                MoveJ Offs(ptPolish,0,0,500),v500,z5,tPolish;
            ENDIF

        DEFAULT:
            !Unknown
            RAISE ERR_TC_SELECTION;

        ENDTEST
        IF dropoffTool THEN
        MoveJ pHome,vMax,fine,tTCMaster;
        ENDIF

    ERROR
        RAISE ;

    ENDPROC

    FUNC num PointToPointDist(num px,num py,num x1,num y1)
        !Used to check if point is within helicopter blades

        VAR num Dist;

        Dist:=Sqrt((x1-px)*(x1-px)+(y1-py)*(y1-py));
        RETURN Dist;
    ENDFUNC

    FUNC num HighestArray(num count)
        !Used to determine highest height offset
        VAR num j;
        VAR num HighestValue;
        HighestValue:=HeliZArray{1};
        FOR j FROM 1 TO count DO
            IF HeliZArray{j}>HighestValue THEN
                HighestValue:=HeliZArray{j};
            ENDIF
        ENDFOR
        IF PreviousHighest>HighestValue THEN
            PreviousHighest:=HighestValue;
            RETURN PreviousHighest;
        ELSEIF HighestValue<=-30 THEN
            PreviousHighest:=HighestValue;
            RETURN 0;
        ELSE
            PreviousHighest:=HighestValue;
            RETURN HighestValue;
        ENDIF

    ENDFUNC

    PROC HeliZ(num x1,num y1,bool ResetZArray)
        !Determines height offsets for helicopter movements
        VAR num CloseYPos;
        x1:=Abs(x1);
        IF ResetZArray=TRUE THEN
            HeliZArrayCounter:=1;
            FOR i FROM 1 TO DIM(HeliZArray,1) DO
                HeliZArray{i}:=-50;
            ENDFOR
        ENDIF

        FOR i FROM 1 TO 17 DO
            FOR j FROM 1 TO 4 DO
                IF PointToPointDist(x1,y1,BedZpos{j,i,1},BedZpos{j,i,2})<=HeliBladeWidth/2 THEN
                    HeliZArray{HeliZArrayCounter}:=BedZreads{j,i};
                    Incr HeliZArrayCounter;
                ENDIF
            ENDFOR
        ENDFOR

    ENDPROC

    PROC PlotBedGrid(num Xcord1,num Ycord1,num ZOffset)
        !Used by BedGridPlotter for Z datum
        Plotterp1.trans:=[Xcord1,Ycord1,200+ZOffset];
        !+46

        IF Plotterp1.trans.y>0 THEN
            IF Plotterp1.trans.y<(abs(tPlotter.tframe.trans.x)-10) THEN
                PlotterZOri:=ACos(Plotterp1.trans.y/abs(tPlotter.tframe.trans.x));
                IF PlotterZOri>PlotA6Max THEN
                    PlotterZOri:=90;
                ENDIF
                Plotterp1.rot:=OrientZYX(-90+PlotterZOri,0,180);
            ELSE
                PlotterZOri:=0;
                Plotterp1.rot:=OrientZYX(-90,0,180);
            ENDIF
        ELSE
            RAISE ERR_PLOT_POS;
        ENDIF

        IF PlotterP1.trans.y>(abs(tPlotter.tframe.trans.x)+250) THEN
            Plotterp1.extax:=[(Plotterp1.trans.x+Bed1.uframe.trans.x),9E+09,9E+09,9E+09,9E+09,9E+09];
        ELSE
            Plotterp1.extax:=[(Plotterp1.trans.x+Bed1.uframe.trans.x+1000+Abs(tPlotter.tframe.trans.x*Sin(PlotterZOri))),9E+09,9E+09,9E+09,9E+09,9E+09];
        ENDIF

        IF Plotterp1.extax.eax_a>10150 THEN
            Plotterp1.extax.eax_a:=10100;
        ENDIF

        IF Plotterp1.extax.eax_a<0 THEN
            Plotterp1.extax.eax_a:=0;
        ENDIF

        vPlotter:=[100,15,2000,15];

        MoveL Plotterp1,v300,zPlotter,tTCMaster\WObj:=Bed1Wyong;

    ENDPROC

    PROC BedGridPlotter()
        !Get Z datum offset
        FOR k FROM 7 TO 19 DO
            !Move x
            FOR j FROM 4 TO 9 DO
                !Move y

                PlotBedGrid(k*XGridSpacing+100),(j*YGridSpacing+100),Bed1Zread{10-j,(k+1)};
                WaitTime\inpos,0.1;

            ENDFOR

        ENDFOR

    ENDPROC

    PROC MoveGridDatum()
        !Sweep across bed maintaining Z height through offsets
        FOR j FROM 9 TO 4 DO
            FOR k FROM 11 TO 1 DO
                !Move x
                PlotBedGrid(k*XGridSpacing+100),(j*YGridSpacing+100),Bed1Zread{10-j,(k+1)};
            ENDFOR
        ENDFOR
    ENDPROC


    PROC VacuumBed()

        VAR num VacOverlap:=-400;
        UpdateToolNum;
        IF ToolNum<>5 THEN
            Home TRUE;
            Vac_Pickup;
        ELSE
            CurrentJoints:=CJointT();
            CurrentPos:=CalcRobT(CurrentJoints,tVac\WObj:=Bed1Wyong);
            IF CurrentPos.trans.x<0 AND (CurrentPos.trans.z<150) THEN
                MoveL Offs(CurrentPos,0,0,(150-CurrentPos.trans.z)),v500,z5,tVac\WObj:=Bed1Wyong;
            ELSEIF (CurrentPos.trans.z<700) THEN
                MoveL Offs(CurrentPos,0,0,(700-CurrentPos.trans.z)),v500,z5,tVac\WObj:=Bed1Wyong;
            ENDIF
        ENDIF

        pTemp:=pVacStart;
        pTemp2:=pVacStart;
        pTemp2.trans.x:=pVacStart2.trans.x;
        pTemp2.extax.eax_a:=pVacStart2.extax.eax_a;

        Vac_on;
        FOR i FROM 0 TO (Round((pVacStart.trans.y-pVacStart2.trans.y)/(-1*VacOverlap))) DO
            IF pTemp.trans.y+i*VacOverlap>pVacStart2.trans.y THEN
                MoveJ Offs(pTemp,0,i*VacOverlap,150),v500,z5,tVac\WObj:=Bed1Wyong;
                MoveL Offs(pTemp,0,i*VacOverlap,0),v50,z5,tVac\WObj:=Bed1Wyong;
                MoveL Offs(pTemp2,0,i*VacOverlap,0),v100,z5,tVac\WObj:=Bed1Wyong;
                MoveL Offs(pTemp2,0,i*VacOverlap,150),v50,fine,tVac\WObj:=Bed1Wyong;
            ENDIF
        ENDFOR

        Vac_off;

        CurrentJoints:=CJointT();
        CurrentPos:=CalcRobT(CurrentJoints,tVac\WObj:=wobj0);
        MoveL Offs(CurrentPos,0,0,800-CurrentPos.trans.z),v100,z5,tVac\WObj:=wobj0;

    ENDPROC

    PROC JointPositions()

        VAR num PolishOverlap:=450;
        pPolTemp:=pPolStart1;
        pPolTemp2:=pPolStart1;
        pPolTemp2.extax.eax_a:=pPolStart1.extax.eax_a-7500;
        pPolTemp2.trans.x:=-7500;

        pPolTemp.rot:=pPolStart1.rot;
        pPolTemp2.rot:=pPolStart1.rot;

        pPolTemp2.rot:=pPolStart2.rot;
        pPolTemp2.extax.eax_a:=pPolStart1.extax.eax_a-8500;
        CurrentJoints5:=CJointT();
        CurrentJoints6:=CalcJointT(Offs(pPolTemp2,50,(1+1)*PolishOverlap,40),tPolish\WObj:=Bed1Wyong);

    ENDPROC


    PROC RobbiePlot()

        ! !Write R
        !PlotLine 6900,1000, 6900,2000;
        !PlotArc 6900,2000,6650,1750,6900,1500;
        !PlotLine 6900,1500,6650,1000;

        !!Write O
        !PlotArc 6300,2000, 6050,1500,6300,1000;
        !PlotArc 6300,1000, 6550,1500,6300,2000;

        !!Write B
        !PlotLine 5700,1000, 5700,2000;
        !PlotArc 5700,2000,5450,1750,5700,1500;
        !PlotArc 5700,1500,5450,1250,5700,1000;

        !!Write B
        !PlotLine 5100,1000, 5100,2000;
        !PlotArc 5100,2000,4850,1750,5100,1500;
        !PlotArc 5100,1500,4850,1250,5100,1000;

        !!Write I
        !PlotLine 4500,1000, 4500,2000;

        !!Write E
        !PlotLine 3900,1000, 3900,2000;
        !PlotLine 3900,2000, 3400,2000;
        !PlotLine 3900,1500, 3400,1500;
        !PlotLine 3900,1000, 3400,1000;

        !formbox
        PlotRect 2000,500,2000,3500,6000,3500,6000,500;
        !Ferrule
        WaitTime\inpos,0.1;
        PlotCirc 2250,750,(PlotCircleD/2);
        PlotLine(2250-PlotCircleD/2-CrossHairExt),750,(2250+PlotCircleD/2+CrossHairExt),750;
        PlotLine 2250,(750-PlotCircleD/2-CrossHairExt),2250,(750+PlotCircleD/2+CrossHairExt);
        !Ferrule
        WaitTime\inpos,0.1;
        PlotCirc 2250,3250,(PlotCircleD/2);
        PlotLine(2250-PlotCircleD/2-CrossHairExt),3250,(2250+PlotCircleD/2+CrossHairExt),3250;
        PlotLine 2250,(3250-PlotCircleD/2-CrossHairExt),2250,(3250+PlotCircleD/2+CrossHairExt);
        !Grout tube Casee 4
        WaitTime\inpos,0.1;
        iCoord1x:=6000;
        iCoord1y:=2000;
        iAngle:=0;
        PlotRect iCoord1x-GroutWidth/2*Sin(iAngle)-GroutHeight*Cos(iAngle),iCoord1y+GroutHeight*Sin(iAngle)-GroutWidth/2*Cos(iAngle),iCoord1x+GroutWidth/2*Sin(iAngle)-GroutHeight*Cos(iAngle),iCoord1y+GroutHeight*Sin(iAngle)+GroutWidth/2*Cos(iAngle),iCoord1x+GroutWidth/2*Sin(iAngle),iCoord1y+GroutWidth/2*Cos(iAngle),iCoord1x-GroutWidth/2*Sin(iAngle),iCoord1y-GroutWidth/2*Cos(iAngle);

        !Lifting points 180 angle
        WaitTime\inpos,0.1;
        TriangleAngle:=180;
        iCoord1x:=5000;
        iCoord1y:=3500;
        PlotLine iCoord1x-TriangleHeight*Sin(TriangleAngle),iCoord1y-TriangleHeight*Cos(TriangleAngle),iCoord1x-TriangleBase/2*Cos(TriangleAngle),iCoord1y+TriangleBase/2*Sin(TriangleAngle);
        PlotLine iCoord1x-TriangleBase/2*Cos(TriangleAngle),iCoord1y+TriangleBase/2*Sin(TriangleAngle),iCoord1x+TriangleBase/2*Cos(TriangleAngle),iCoord1y-TriangleBase/2*Sin(TriangleAngle);
        PlotLine iCoord1x+TriangleBase/2*Cos(TriangleAngle),iCoord1y-TriangleBase/2*Sin(TriangleAngle),iCoord1x-TriangleHeight*Sin(TriangleAngle),iCoord1y-TriangleHeight*Cos(TriangleAngle);
        !Lifting points 180 angle
        WaitTime\inpos,0.1;
        TriangleAngle:=180;
        iCoord1x:=3000;
        iCoord1y:=3500;
        PlotLine iCoord1x-TriangleHeight*Sin(TriangleAngle),iCoord1y-TriangleHeight*Cos(TriangleAngle),iCoord1x-TriangleBase/2*Cos(TriangleAngle),iCoord1y+TriangleBase/2*Sin(TriangleAngle);
        PlotLine iCoord1x-TriangleBase/2*Cos(TriangleAngle),iCoord1y+TriangleBase/2*Sin(TriangleAngle),iCoord1x+TriangleBase/2*Cos(TriangleAngle),iCoord1y-TriangleBase/2*Sin(TriangleAngle);
        PlotLine iCoord1x+TriangleBase/2*Cos(TriangleAngle),iCoord1y-TriangleBase/2*Sin(TriangleAngle),iCoord1x-TriangleHeight*Sin(TriangleAngle),iCoord1y-TriangleHeight*Cos(TriangleAngle);

        Plotter_Dropoff;

    ENDPROC

    PROC PolishDemo()
        UpdateToolNum;
        IF ToolNum<>6 THEN
            Home TRUE;
            Polish_Pickup;
        ELSE
            CurrentJoints:=CJointT();
            CurrentPos:=CalcRobT(CurrentJoints,tPolish\WObj:=wobj0);
            IF CurrentPos.trans.z<600 THEN
                MoveL Offs(CurrentPos,0,0,(600-CurrentPos.trans.z)),v500,z5,tPolish;
            ENDIF
        ENDIF
        MoveJ pPolHome,v500,z5,tPolish;
        pPolTemp:=pPolStart1;
        pPolTemp2:=pPolStart1;
        pPolTemp2.extax.eax_a:=pPolStart1.extax.eax_a-7500;
        pPolTemp2.trans.x:=-7500;
        pPolTemp.rot:=pPolStart1.rot;
        pPolTemp2.rot:=pPolStart1.rot;
        FCCalib PolishLoad;
        pPolTemp.extax.eax_a:=pPolStart1.extax.eax_a;
        MoveJ Offs(pPolTemp,0,0,100),v500,z5,tPolish\WObj:=Bed1Wyong;
        Pol_on;
        MoveL Offs(pPolTemp,0,0,50),v100,fine,tPolish\WObj:=Bed1Wyong;
        myForceVector:=FCGetForce(\Tool:=tPolish);
        FCPress1LStart Offs(pPolTemp,-25,0,55),v10,\Fz:=120,15,\ForceChange:=50\PosSupvDist:=125,z5,tPolish\WObj:=Bed1Wyong;
        pPolTemp2.extax.eax_a:=pPolStart2.extax.eax_a-300;
        FCPressL Offs(pPolTemp2,-300,0,-15),v100,130,fine,tPolish\WObj:=Bed1Wyong;
        FCPressEnd Offs(pPolTemp2,-300,0,75),v50,\DeactOnly,tPolish\WObj:=Bed1Wyong;
        CurrentJoints:=CJointT();
        CurrentPos:=CalcRobT(CurrentJoints,tPolish\WObj:=Bed1Wyong);
        MoveJ Offs(Reltool(CurrentPos,0,0,-100),0,450,0),v100,fine,tPolish\WObj:=Bed1Wyong;
        Pol_off;
        Polish_Dropoff;
    ENDPROC



    PROC BedGrid()

        !        MoveJ Offs(p10Maps,500*(1-1)+2000*(1-1),650*(1-1),50),v500,z5,tTCMaster\WObj:=Bed1Wyong;
        !        MoveL Offs(p10Maps,500*(1-1)+2000*(1-1),650*(1-1),0),v500,fine,tTCMaster\WObj:=Bed1Wyong;
        !        Stop;
        !        MoveL Offs(p10Maps,500*(1-1)+2000*(1-1),650*(1-1),50),v500,z5,tTCMaster\WObj:=Bed1Wyong;
        !        Stop;

        FOR i FROM 1 TO 5 DO
            !Move EAX
            FOR k FROM 1 TO 4 DO
                !Move x
                FOR j FROM 1 TO 4 DO
                    !Move y
                    IF 500*(k-1)+2000*(i-1)<8001 THEN
                        p10maps.extax.eax_a:=Bed1Wyong.uframe.trans.x+p10Maps.trans.x-500*(k-1)-2000*(i-1);
                        IF p10maps.extax.eax_a>10150 THEN
                            p10maps.extax.eax_a:=10100;
                        ENDIF
                        IF p10maps.extax.eax_a<1000 THEN
                            p10maps.extax.eax_a:=1000;
                        ENDIF

                        !MoveJ Offs(p10Maps,-500*(k-1)-2000*(i-1),650*(j-1),50),v500,z5,tTCMaster\WObj:=Bed1Wyong;
                        !MoveL Offs(p10Maps,-500*(k-1)-2000*(i-1),650*(j-1),0),v500,fine,tTCMaster\WObj:=Bed1Wyong;
                        !TPReadNum BedZread,"Enter Z reading";
                        !BedZreads{5-j,((i-1)*4+k)}:=BedZread;
                        BedZpos{5-j,((i-1)*4+k),1}:=p10Maps.trans.x-500*(k-1)-2000*(i-1);
                        BedZpos{5-j,((i-1)*4+k),2}:=p10maps.trans.y+650*(j-1);
                        !MoveL Offs(p10Maps,-500*(k-1)-2000*(i-1),650*(j-1),50),v500,z5,tTCMaster\WObj:=Bed1Wyong;
                    ENDIF

                ENDFOR
            ENDFOR
        ENDFOR
        Stop;

    ENDPROC


    PROC ClearBedZ()

        FOR i FROM 1 TO 4 DO
            !Move EAX
            FOR k FROM 1 TO 24 DO
                !Move x
                BedZreads{i,k}:=0;
                BedZpos{i,k,1}:=0;
                BedZpos{i,k,2}:=0;
            ENDFOR
        ENDFOR

    ENDPROC




    PROC BHTestTask()
        TPErase;
        TPWrite "BH Test Task";
        TPWrite "Press Play to confirm and start task";
        Stop;

        TPErase;
        TPWrite "Starting BH Test Task...";

        Heli_Pickup;
        MoveJ Offs(ptHeli,0,0,1000),v500,fine,tHeli;
        TPWrite "Helicopter tool at 1000mm above pickup";
        WaitTime 2;

        Heli_Dropoff;
        TPWrite "Helicopter tool dropped off";

        Polish_Pickup;
        MoveJ Offs(ptPolish,0,0,1000),v500,fine,tPolish;
        TPWrite "Polisher tool at 1000mm above pickup";
        WaitTime 2;

        Polish_Dropoff;
        TPWrite "Polisher tool dropped off";

        Home TRUE;
        TPWrite "BH Test Task Complete";

    ERROR
        RAISE ;
    ENDPROC



    PROC Datum()
        ! Datum - draws small circle at Bed1Wyong origin (0,0)
        ! Generated by Onyx Toolpath Generator
        VAR robtarget pDatumCenter;
        VAR robtarget pDatumCircle;
        VAR num DatumZ:=300;
        VAR num DatumRadius:=100;
        VAR num SafeZ:=500;
        VAR num i;

        UpdateToolNum;
        TPWrite "Datum: ToolNum=" \Num:=ToolNum;
        IF ToolNum<>4 THEN
            TPWrite "No plotter! Will pickup plotter.";
            Stop;
            Home TRUE;
            Plotter_Pickup;
        ELSE
            CurrentJoints:=CJointT();
            CurrentPos:=CalcRobT(CurrentJoints,tPlotter\WObj:=wobj0);
            IF CurrentPos.trans.z<600 THEN
                MoveL Offs(CurrentPos,0,0,(600-CurrentPos.trans.z)),v500,z5,tPlotter;
            ENDIF
        ENDIF

        ConfL\Off;
        ConfJ\Off;

        pDatumCenter:=[[0,0,DatumZ],[0,0,1,0],[0,0,0,0],[0,9E+09,9E+09,9E+09,9E+09,9E+09]];
        pDatumCenter.rot:=OrientZYX(-90,0,180);
        pDatumCenter.extax.eax_a:=6500;

        TPWrite "Datum: Drawing circle at origin";
        TPWrite "Press Play to continue";
        Stop;

        pDatumCircle:=pDatumCenter;
        pDatumCircle.trans.z:=SafeZ;
        MoveJ pDatumCircle,v500,z5,tPlotter\WObj:=Bed1Wyong;

        pDatumCircle.trans.x:=DatumRadius;
        pDatumCircle.trans.z:=DatumZ;
        MoveJ pDatumCircle,v500,z5,tPlotter\WObj:=Bed1Wyong;

        FOR i FROM 1 TO 8 DO
            pDatumCircle.trans.x:=DatumRadius*Cos(i*45);
            pDatumCircle.trans.y:=DatumRadius*Sin(i*45);
            MoveJ pDatumCircle,v100,fine,tPlotter\WObj:=Bed1Wyong;
        ENDFOR

        pDatumCircle.trans.x:=0;
        pDatumCircle.trans.y:=0;
        pDatumCircle.trans.z:=DatumZ;
        MoveJ pDatumCircle,v100,fine,tPlotter\WObj:=Bed1Wyong;

        TPWrite "Plotter at datum center (0,0)";
        TPWrite "Press Play to return tool";
        Stop;

        pDatumCircle.trans.z:=SafeZ;
        MoveJ pDatumCircle,v500,z5,tPlotter\WObj:=Bed1Wyong;

        ConfL\On;
        ConfJ\On;

        Plotter_Dropoff;
        Home TRUE;

        TPWrite "Datum Complete";
    ERROR
        RAISE;
    ENDPROC

    PROC RequestAccessCheck()

        IF TestDI (PN_DI_08) AND (TestDI (PN_DI_09) = FALSE) THEN
            Home TRUE;
            SetDO PN_DO_08,1;
        ENDIF
            IF TestDI (PN_DI_09)  THEN
                SetDO PN_DO_10,0;
                Home FALSE;
                SetDO PN_DO_09, 1;
            ENDIF



    ENDPROC
    PROC Automoving()

        MoveJ pVSautoTest4, v500, z10, tTCmaster;
        MoveJ pVSautoTest3, v500, z10, tTCmaster;

    ENDPROC


    ! ========== PY2 GENERATED PROCEDURES ==========
    ! Generated: 10-mar_08:05
    ! Do not edit manually - regenerate via web interface


    PROC MainMenu()
        VAR num iTask;
        TPErase;
        TPReadNum iTask,"1:Home,2:Py2_10-mar_08:05";
        TEST iTask
        CASE 1:
            Home TRUE;
        CASE 2:
            Py2Main;
        DEFAULT:
            RAISE ERR_INVALID_INPUT;
        ENDTEST
    ERROR
        RAISE;
    ENDPROC


    PROC Py2Main()
        ! Py2Main - Python-generated tools menu
        ! Generated: 10-mar_08:05

        VAR num iChoice;

        TPErase;
        TPWrite "=== Py2 Tools (10-mar_08:05) ===";
        TPWrite "Panel X: " \Num:=6000;
        TPWrite "Panel Y: " \Num:=3500;
        TPReadNum iChoice,"1:Heli,2:Polish,3:Vac,4:Pan,5:Screed,6:BedClean";

        TEST iChoice
        CASE 1:
            Py2Heli;
        CASE 2:
            Py2Polish;
        CASE 3:
            Py2Vac;
        CASE 4:
            Py2Pan;
        CASE 5:
            Py2VS;
        CASE 6:
            SeqBedClean;
        DEFAULT:
            TPWrite "Invalid choice";
        ENDTEST
    ENDPROC


    PROC Py2Heli()
        ! Py2Heli - Generated by Onyx Tool Class
        ! Workzone: panel
        ! Area: (530,300) to (5930,1550)
        ! Z = 455mm
        ! Step: 200mm

        VAR robtarget pCurrent;
        VAR jointtarget CurrentJoints;
        VAR robtarget CurrentPos;
        VAR num WorkZ:=455;
        VAR num SafeZ:=655;
        VAR num CurrentX:=0;
        VAR num CurrentY:=0;
        VAR speeddata vTravel:=[100,500,5000,1000];
        VAR num TrackMin:=-300;
        VAR num TrackMax:=10050;
        VAR num CalcTrack:=0;
        VAR num HeliForce:=0;
        VAR bool bFCActive:=FALSE;
        VAR fcforcevector myForceVector;

        TPWrite "========================================";
        TPWrite "Py2Heli: Starting";
        TPWrite "========================================";
        TPWrite "Workzone: panel";
        TPWrite "WorkZ=" \Num:=WorkZ;

        ! Get tool if needed
        UpdateToolNum;
        IF ToolNum<>2 THEN
            TPWrite "Py2Heli: Getting tool...";
            Home TRUE;
            Heli_Pickup;
        ELSE
            CurrentJoints:=CJointT();
            CurrentPos:=CalcRobT(CurrentJoints,tHeli\WObj:=wobj0);
            IF (CurrentPos.trans.x)>8000 AND CurrentPos.trans.z<400 THEN
                MoveL Offs(CurrentPos,0,0,(400-CurrentPos.trans.z)),v100,z5,tHeli;
            ENDIF
        ENDIF

        ! Set blade pitch angle
        HeliBlade_Angle 7;

        ! Start blade rotation
        HeliBladeSpeed 80,"REV";
        WaitTime 2;

        ! ========================================
        ! Pattern Execution: 9 points
        ! ========================================

        ! Point 1: (780, 1300) [rapid]
        CurrentX:=780;
        CurrentY:=1300;
        pCurrent.trans:=[-1*CurrentX,CurrentY,SafeZ];
        pCurrent.rot:=OrientZYX(0,0,180);
        pCurrent.robconf:=[1,0,-2,0];
        CalcTrack:=Bed1Wyong.uframe.trans.x+pCurrent.trans.x;
        IF CurrentY<1000 THEN CalcTrack:=CalcTrack+1200; ENDIF
        IF CalcTrack<TrackMin THEN CalcTrack:=TrackMin; ENDIF
        IF CalcTrack>TrackMax THEN CalcTrack:=TrackMax; ENDIF
        pCurrent.extax:=[CalcTrack,9E+09,9E+09,9E+09,9E+09,9E+09];
        MoveJ pCurrent,v500,z5,tHeli\WObj:=Bed1Wyong;

        ! Descend to work height
        pCurrent.trans.z:=WorkZ;
        MoveL pCurrent,v100,fine,tHeli\WObj:=Bed1Wyong;

        ! Point 2: (5680, 1300) [work]
        CurrentX:=5680;
        CurrentY:=1300;
        pCurrent.trans:=[-1*CurrentX,CurrentY,WorkZ];
        pCurrent.rot:=OrientZYX(0,0,180);
        pCurrent.robconf:=[1,0,-2,0];
        CalcTrack:=Bed1Wyong.uframe.trans.x+pCurrent.trans.x;
        IF CurrentY<1000 THEN CalcTrack:=CalcTrack+1200; ENDIF
        IF CalcTrack<TrackMin THEN CalcTrack:=TrackMin; ENDIF
        IF CalcTrack>TrackMax THEN CalcTrack:=TrackMax; ENDIF
        pCurrent.extax:=[CalcTrack,9E+09,9E+09,9E+09,9E+09,9E+09];
        MoveL pCurrent,vTravel,fine,tHeli\WObj:=Bed1Wyong;

        ! Point 3: (5680, 550) [work]
        CurrentX:=5680;
        CurrentY:=550;
        pCurrent.trans:=[-1*CurrentX,CurrentY,WorkZ];
        pCurrent.rot:=OrientZYX(0,0,180);
        pCurrent.robconf:=[1,0,-2,0];
        CalcTrack:=Bed1Wyong.uframe.trans.x+pCurrent.trans.x;
        IF CurrentY<1000 THEN CalcTrack:=CalcTrack+1200; ENDIF
        IF CalcTrack<TrackMin THEN CalcTrack:=TrackMin; ENDIF
        IF CalcTrack>TrackMax THEN CalcTrack:=TrackMax; ENDIF
        pCurrent.extax:=[CalcTrack,9E+09,9E+09,9E+09,9E+09,9E+09];
        MoveL pCurrent,vTravel,fine,tHeli\WObj:=Bed1Wyong;

        ! Point 4: (780, 550) [work]
        CurrentX:=780;
        CurrentY:=550;
        pCurrent.trans:=[-1*CurrentX,CurrentY,WorkZ];
        pCurrent.rot:=OrientZYX(0,0,180);
        pCurrent.robconf:=[1,0,-2,0];
        CalcTrack:=Bed1Wyong.uframe.trans.x+pCurrent.trans.x;
        IF CurrentY<1000 THEN CalcTrack:=CalcTrack+1200; ENDIF
        IF CalcTrack<TrackMin THEN CalcTrack:=TrackMin; ENDIF
        IF CalcTrack>TrackMax THEN CalcTrack:=TrackMax; ENDIF
        pCurrent.extax:=[CalcTrack,9E+09,9E+09,9E+09,9E+09,9E+09];
        MoveL pCurrent,vTravel,fine,tHeli\WObj:=Bed1Wyong;

        ! Point 5: (780, 1100) [work]
        CurrentX:=780;
        CurrentY:=1100;
        pCurrent.trans:=[-1*CurrentX,CurrentY,WorkZ];
        pCurrent.rot:=OrientZYX(0,0,180);
        pCurrent.robconf:=[1,0,-2,0];
        CalcTrack:=Bed1Wyong.uframe.trans.x+pCurrent.trans.x;
        IF CurrentY<1000 THEN CalcTrack:=CalcTrack+1200; ENDIF
        IF CalcTrack<TrackMin THEN CalcTrack:=TrackMin; ENDIF
        IF CalcTrack>TrackMax THEN CalcTrack:=TrackMax; ENDIF
        pCurrent.extax:=[CalcTrack,9E+09,9E+09,9E+09,9E+09,9E+09];
        MoveL pCurrent,vTravel,fine,tHeli\WObj:=Bed1Wyong;

        ! Point 6: (5480, 1100) [work]
        CurrentX:=5480;
        CurrentY:=1100;
        pCurrent.trans:=[-1*CurrentX,CurrentY,WorkZ];
        pCurrent.rot:=OrientZYX(0,0,180);
        pCurrent.robconf:=[1,0,-2,0];
        CalcTrack:=Bed1Wyong.uframe.trans.x+pCurrent.trans.x;
        IF CurrentY<1000 THEN CalcTrack:=CalcTrack+1200; ENDIF
        IF CalcTrack<TrackMin THEN CalcTrack:=TrackMin; ENDIF
        IF CalcTrack>TrackMax THEN CalcTrack:=TrackMax; ENDIF
        pCurrent.extax:=[CalcTrack,9E+09,9E+09,9E+09,9E+09,9E+09];
        MoveL pCurrent,vTravel,fine,tHeli\WObj:=Bed1Wyong;

        ! Point 7: (5480, 750) [work]
        CurrentX:=5480;
        CurrentY:=750;
        pCurrent.trans:=[-1*CurrentX,CurrentY,WorkZ];
        pCurrent.rot:=OrientZYX(0,0,180);
        pCurrent.robconf:=[1,0,-2,0];
        CalcTrack:=Bed1Wyong.uframe.trans.x+pCurrent.trans.x;
        IF CurrentY<1000 THEN CalcTrack:=CalcTrack+1200; ENDIF
        IF CalcTrack<TrackMin THEN CalcTrack:=TrackMin; ENDIF
        IF CalcTrack>TrackMax THEN CalcTrack:=TrackMax; ENDIF
        pCurrent.extax:=[CalcTrack,9E+09,9E+09,9E+09,9E+09,9E+09];
        MoveL pCurrent,vTravel,fine,tHeli\WObj:=Bed1Wyong;

        ! Point 8: (980, 750) [work]
        CurrentX:=980;
        CurrentY:=750;
        pCurrent.trans:=[-1*CurrentX,CurrentY,WorkZ];
        pCurrent.rot:=OrientZYX(0,0,180);
        pCurrent.robconf:=[1,0,-2,0];
        CalcTrack:=Bed1Wyong.uframe.trans.x+pCurrent.trans.x;
        IF CurrentY<1000 THEN CalcTrack:=CalcTrack+1200; ENDIF
        IF CalcTrack<TrackMin THEN CalcTrack:=TrackMin; ENDIF
        IF CalcTrack>TrackMax THEN CalcTrack:=TrackMax; ENDIF
        pCurrent.extax:=[CalcTrack,9E+09,9E+09,9E+09,9E+09,9E+09];
        MoveL pCurrent,vTravel,fine,tHeli\WObj:=Bed1Wyong;

        ! Point 9: (980, 900) [work]
        CurrentX:=980;
        CurrentY:=900;
        pCurrent.trans:=[-1*CurrentX,CurrentY,WorkZ];
        pCurrent.rot:=OrientZYX(0,0,180);
        pCurrent.robconf:=[1,0,-2,0];
        CalcTrack:=Bed1Wyong.uframe.trans.x+pCurrent.trans.x;
        IF CurrentY<1000 THEN CalcTrack:=CalcTrack+1200; ENDIF
        IF CalcTrack<TrackMin THEN CalcTrack:=TrackMin; ENDIF
        IF CalcTrack>TrackMax THEN CalcTrack:=TrackMax; ENDIF
        pCurrent.extax:=[CalcTrack,9E+09,9E+09,9E+09,9E+09,9E+09];
        MoveL pCurrent,vTravel,fine,tHeli\WObj:=Bed1Wyong;

        ! Stop blade rotation
        HeliBladeSpeed 0,"FWD";
        WaitTime 1;

        ! Lift to safe height
        CurrentJoints:=CJointT();
        CurrentPos:=CalcRobT(CurrentJoints,tHeli\WObj:=Bed1Wyong);
        MoveL Offs(CurrentPos,0,0,200),v200,z5,tHeli\WObj:=Bed1Wyong;

        ! Return tool and go home
        TPWrite "Py2Heli: Dropping off tool...";
        Heli_Dropoff;
        Home FALSE;

        TPWrite "========================================";
        TPWrite "Py2Heli: COMPLETE";
        TPWrite "========================================";

    ERROR
        HeliBladeSpeed 0,"FWD";
        IF bFCActive THEN
            FCPressEnd Offs(CurrentPos,0,0,100),v50,\DeactOnly,tHeli\WObj:=Bed1Wyong;
        ENDIF
        RAISE;
    ENDPROC

    PROC Py2Polish()
        ! Py2Polish - Generated by Onyx Tool Class
        ! Workzone: bed
        ! Area: (100,100) to (8150,1750)
        ! Z = 305mm
        ! Step: 350mm

        VAR robtarget pCurrent;
        VAR jointtarget CurrentJoints;
        VAR robtarget CurrentPos;
        VAR num WorkZ:=305;
        VAR num SafeZ:=505;
        VAR num CurrentX:=0;
        VAR num CurrentY:=0;
        VAR speeddata vTravel:=[500,500,5000,1000];
        VAR num TrackMin:=-300;
        VAR num TrackMax:=10050;
        VAR num CalcTrack:=0;
        VAR bool bFCActive:=FALSE;
        VAR fcboxvol fc_supv_box:=[-10000,10000,-10000,10000,-10000,10000];

        TPWrite "========================================";
        TPWrite "Py2Polish: Starting";
        TPWrite "========================================";
        TPWrite "Workzone: bed";
        TPWrite "WorkZ=" \Num:=WorkZ;

        ! Get tool if needed
        UpdateToolNum;
        IF ToolNum<>6 THEN
            TPWrite "Py2Polish: Getting tool...";
            Home TRUE;
            Polish_Pickup;
        ELSE
            CurrentJoints:=CJointT();
            CurrentPos:=CalcRobT(CurrentJoints,tPolish\WObj:=wobj0);
            IF (CurrentPos.trans.x)>8000 AND CurrentPos.trans.z<400 THEN
                MoveL Offs(CurrentPos,0,0,(400-CurrentPos.trans.z)),v100,z5,tPolish;
            ENDIF
        ENDIF

        ! ========================================
        ! Polisher Pattern Execution: 60 points
        ! Force Control: ENABLED
        ! ========================================

        ! Rapid: (100, 1750)
        CurrentX:=100;
        CurrentY:=1750;
        pCurrent.trans:=[-1*CurrentX,CurrentY,SafeZ];
        pCurrent.rot:=OrientZYX(0,0,180);
        pCurrent.robconf:=[0,0,0,0];
        CalcTrack:=Bed1Wyong.uframe.trans.x+pCurrent.trans.x;
        IF CurrentY<1000 THEN CalcTrack:=CalcTrack+1200; ENDIF
        IF CalcTrack<TrackMin THEN CalcTrack:=TrackMin; ENDIF
        IF CalcTrack>TrackMax THEN CalcTrack:=TrackMax; ENDIF
        pCurrent.extax:=[CalcTrack,9E+09,9E+09,9E+09,9E+09,9E+09];
        MoveJ pCurrent,v500,z5,tPolish\WObj:=Bed1Wyong;

        ! Lower to 250mm above work surface
        pCurrent.trans.z:=WorkZ+250;
        MoveL pCurrent,v100,fine,tPolish\WObj:=Bed1Wyong;
        WaitTime\inpos,0.1;

        ! Force control calibration (must be done with motor OFF)
        FCCalib PolishLoad;

        ! Turn on polisher motor
        Pol_on;

        ! Lower to 80mm above work surface
        pCurrent.trans.z:=WorkZ+80;
        MoveL pCurrent,v100,fine,tPolish\WObj:=Bed1Wyong;
        WaitTime\inpos,0.1;

        ! Start force control - pressing from ~50mm above work surface
        pCurrent.trans.z:=WorkZ+50;
        FCPress1LStart pCurrent,v20,\Fz:=300,15,\ForceChange:=150\PosSupvDist:=100,z5,tPolish\WObj:=Bed1Wyong;
        bFCActive:=TRUE;

        ! Work point 1: (8150, 1750) [work]
        CurrentX:=8150;
        CurrentY:=1750;
        pCurrent.trans:=[-1*CurrentX,CurrentY,WorkZ];
        pCurrent.robconf:=[0,0,0,0];
        CalcTrack:=Bed1Wyong.uframe.trans.x+pCurrent.trans.x;
        IF CurrentY<1000 THEN CalcTrack:=CalcTrack+1200; ENDIF
        IF CalcTrack<TrackMin THEN CalcTrack:=TrackMin; ENDIF
        IF CalcTrack>TrackMax THEN CalcTrack:=TrackMax; ENDIF
        pCurrent.extax:=[CalcTrack,9E+09,9E+09,9E+09,9E+09,9E+09];
        FCPressL pCurrent,v500,150,fine,tPolish\WObj:=Bed1Wyong;

        ! Work point 2: (8150, 1400) [work]
        CurrentX:=8150;
        CurrentY:=1400;
        pCurrent.trans:=[-1*CurrentX,CurrentY,WorkZ];
        pCurrent.robconf:=[0,0,0,0];
        CalcTrack:=Bed1Wyong.uframe.trans.x+pCurrent.trans.x;
        IF CurrentY<1000 THEN CalcTrack:=CalcTrack+1200; ENDIF
        IF CalcTrack<TrackMin THEN CalcTrack:=TrackMin; ENDIF
        IF CalcTrack>TrackMax THEN CalcTrack:=TrackMax; ENDIF
        pCurrent.extax:=[CalcTrack,9E+09,9E+09,9E+09,9E+09,9E+09];
        FCPressL pCurrent,v500,150,fine,tPolish\WObj:=Bed1Wyong;

        ! Work point 3: (100, 1400) [work]
        CurrentX:=100;
        CurrentY:=1400;
        pCurrent.trans:=[-1*CurrentX,CurrentY,WorkZ];
        pCurrent.robconf:=[0,0,0,0];
        CalcTrack:=Bed1Wyong.uframe.trans.x+pCurrent.trans.x;
        IF CurrentY<1000 THEN CalcTrack:=CalcTrack+1200; ENDIF
        IF CalcTrack<TrackMin THEN CalcTrack:=TrackMin; ENDIF
        IF CalcTrack>TrackMax THEN CalcTrack:=TrackMax; ENDIF
        pCurrent.extax:=[CalcTrack,9E+09,9E+09,9E+09,9E+09,9E+09];
        FCPressL pCurrent,v500,150,fine,tPolish\WObj:=Bed1Wyong;

        ! Work point 4: (100, 1050) [work]
        CurrentX:=100;
        CurrentY:=1050;
        pCurrent.trans:=[-1*CurrentX,CurrentY,WorkZ];
        pCurrent.robconf:=[0,0,0,0];
        CalcTrack:=Bed1Wyong.uframe.trans.x+pCurrent.trans.x;
        IF CurrentY<1000 THEN CalcTrack:=CalcTrack+1200; ENDIF
        IF CalcTrack<TrackMin THEN CalcTrack:=TrackMin; ENDIF
        IF CalcTrack>TrackMax THEN CalcTrack:=TrackMax; ENDIF
        pCurrent.extax:=[CalcTrack,9E+09,9E+09,9E+09,9E+09,9E+09];
        FCPressL pCurrent,v500,150,fine,tPolish\WObj:=Bed1Wyong;

        ! Work point 5: (8150, 1050) [work]
        CurrentX:=8150;
        CurrentY:=1050;
        pCurrent.trans:=[-1*CurrentX,CurrentY,WorkZ];
        pCurrent.robconf:=[0,0,0,0];
        CalcTrack:=Bed1Wyong.uframe.trans.x+pCurrent.trans.x;
        IF CurrentY<1000 THEN CalcTrack:=CalcTrack+1200; ENDIF
        IF CalcTrack<TrackMin THEN CalcTrack:=TrackMin; ENDIF
        IF CalcTrack>TrackMax THEN CalcTrack:=TrackMax; ENDIF
        pCurrent.extax:=[CalcTrack,9E+09,9E+09,9E+09,9E+09,9E+09];
        FCPressL pCurrent,v500,150,fine,tPolish\WObj:=Bed1Wyong;

        ! Work point 6: (8150, 700) [work]
        CurrentX:=8150;
        CurrentY:=700;
        pCurrent.trans:=[-1*CurrentX,CurrentY,WorkZ];
        pCurrent.robconf:=[0,0,0,0];
        CalcTrack:=Bed1Wyong.uframe.trans.x+pCurrent.trans.x;
        IF CurrentY<1000 THEN CalcTrack:=CalcTrack+1200; ENDIF
        IF CalcTrack<TrackMin THEN CalcTrack:=TrackMin; ENDIF
        IF CalcTrack>TrackMax THEN CalcTrack:=TrackMax; ENDIF
        pCurrent.extax:=[CalcTrack,9E+09,9E+09,9E+09,9E+09,9E+09];
        FCPressL pCurrent,v500,150,fine,tPolish\WObj:=Bed1Wyong;

        ! Work point 7: (100, 700) [work]
        CurrentX:=100;
        CurrentY:=700;
        pCurrent.trans:=[-1*CurrentX,CurrentY,WorkZ];
        pCurrent.robconf:=[0,0,0,0];
        CalcTrack:=Bed1Wyong.uframe.trans.x+pCurrent.trans.x;
        IF CurrentY<1000 THEN CalcTrack:=CalcTrack+1200; ENDIF
        IF CalcTrack<TrackMin THEN CalcTrack:=TrackMin; ENDIF
        IF CalcTrack>TrackMax THEN CalcTrack:=TrackMax; ENDIF
        pCurrent.extax:=[CalcTrack,9E+09,9E+09,9E+09,9E+09,9E+09];
        FCPressL pCurrent,v500,150,fine,tPolish\WObj:=Bed1Wyong;

        ! Work point 8: (100, 350) [work]
        CurrentX:=100;
        CurrentY:=350;
        pCurrent.trans:=[-1*CurrentX,CurrentY,WorkZ];
        pCurrent.robconf:=[0,0,0,0];
        CalcTrack:=Bed1Wyong.uframe.trans.x+pCurrent.trans.x;
        IF CurrentY<1000 THEN CalcTrack:=CalcTrack+1200; ENDIF
        IF CalcTrack<TrackMin THEN CalcTrack:=TrackMin; ENDIF
        IF CalcTrack>TrackMax THEN CalcTrack:=TrackMax; ENDIF
        pCurrent.extax:=[CalcTrack,9E+09,9E+09,9E+09,9E+09,9E+09];
        FCPressL pCurrent,v500,150,fine,tPolish\WObj:=Bed1Wyong;

        ! Work point 9: (8150, 350) [work]
        CurrentX:=8150;
        CurrentY:=350;
        pCurrent.trans:=[-1*CurrentX,CurrentY,WorkZ];
        pCurrent.robconf:=[0,0,0,0];
        CalcTrack:=Bed1Wyong.uframe.trans.x+pCurrent.trans.x;
        IF CurrentY<1000 THEN CalcTrack:=CalcTrack+1200; ENDIF
        IF CalcTrack<TrackMin THEN CalcTrack:=TrackMin; ENDIF
        IF CalcTrack>TrackMax THEN CalcTrack:=TrackMax; ENDIF
        pCurrent.extax:=[CalcTrack,9E+09,9E+09,9E+09,9E+09,9E+09];
        FCPressL pCurrent,v500,150,fine,tPolish\WObj:=Bed1Wyong;

        ! Work point 10: (8150, 100) [work]
        CurrentX:=8150;
        CurrentY:=100;
        pCurrent.trans:=[-1*CurrentX,CurrentY,WorkZ];
        pCurrent.robconf:=[0,0,0,0];
        CalcTrack:=Bed1Wyong.uframe.trans.x+pCurrent.trans.x;
        IF CurrentY<1000 THEN CalcTrack:=CalcTrack+1200; ENDIF
        IF CalcTrack<TrackMin THEN CalcTrack:=TrackMin; ENDIF
        IF CalcTrack>TrackMax THEN CalcTrack:=TrackMax; ENDIF
        pCurrent.extax:=[CalcTrack,9E+09,9E+09,9E+09,9E+09,9E+09];
        FCPressL pCurrent,v500,150,fine,tPolish\WObj:=Bed1Wyong;

        ! Work point 11: (100, 100) [work]
        CurrentX:=100;
        CurrentY:=100;
        pCurrent.trans:=[-1*CurrentX,CurrentY,WorkZ];
        pCurrent.robconf:=[0,0,0,0];
        CalcTrack:=Bed1Wyong.uframe.trans.x+pCurrent.trans.x;
        IF CurrentY<1000 THEN CalcTrack:=CalcTrack+1200; ENDIF
        IF CalcTrack<TrackMin THEN CalcTrack:=TrackMin; ENDIF
        IF CalcTrack>TrackMax THEN CalcTrack:=TrackMax; ENDIF
        pCurrent.extax:=[CalcTrack,9E+09,9E+09,9E+09,9E+09,9E+09];
        FCPressL pCurrent,v500,150,fine,tPolish\WObj:=Bed1Wyong;

        ! Work point 12: (100, 100) [work]
        CurrentX:=100;
        CurrentY:=100;
        pCurrent.trans:=[-1*CurrentX,CurrentY,WorkZ];
        pCurrent.robconf:=[0,0,0,0];
        CalcTrack:=Bed1Wyong.uframe.trans.x+pCurrent.trans.x;
        IF CurrentY<1000 THEN CalcTrack:=CalcTrack+1200; ENDIF
        IF CalcTrack<TrackMin THEN CalcTrack:=TrackMin; ENDIF
        IF CalcTrack>TrackMax THEN CalcTrack:=TrackMax; ENDIF
        pCurrent.extax:=[CalcTrack,9E+09,9E+09,9E+09,9E+09,9E+09];
        FCPressL pCurrent,v500,150,fine,tPolish\WObj:=Bed1Wyong;

        ! Work point 13: (100, 1750) [work]
        CurrentX:=100;
        CurrentY:=1750;
        pCurrent.trans:=[-1*CurrentX,CurrentY,WorkZ];
        pCurrent.robconf:=[0,0,0,0];
        CalcTrack:=Bed1Wyong.uframe.trans.x+pCurrent.trans.x;
        IF CurrentY<1000 THEN CalcTrack:=CalcTrack+1200; ENDIF
        IF CalcTrack<TrackMin THEN CalcTrack:=TrackMin; ENDIF
        IF CalcTrack>TrackMax THEN CalcTrack:=TrackMax; ENDIF
        pCurrent.extax:=[CalcTrack,9E+09,9E+09,9E+09,9E+09,9E+09];
        FCPressL pCurrent,v500,150,fine,tPolish\WObj:=Bed1Wyong;

        ! Work point 14: (450, 1750) [work]
        CurrentX:=450;
        CurrentY:=1750;
        pCurrent.trans:=[-1*CurrentX,CurrentY,WorkZ];
        pCurrent.robconf:=[0,0,0,0];
        CalcTrack:=Bed1Wyong.uframe.trans.x+pCurrent.trans.x;
        IF CurrentY<1000 THEN CalcTrack:=CalcTrack+1200; ENDIF
        IF CalcTrack<TrackMin THEN CalcTrack:=TrackMin; ENDIF
        IF CalcTrack>TrackMax THEN CalcTrack:=TrackMax; ENDIF
        pCurrent.extax:=[CalcTrack,9E+09,9E+09,9E+09,9E+09,9E+09];
        FCPressL pCurrent,v500,150,fine,tPolish\WObj:=Bed1Wyong;

        ! Work point 15: (450, 100) [work]
        CurrentX:=450;
        CurrentY:=100;
        pCurrent.trans:=[-1*CurrentX,CurrentY,WorkZ];
        pCurrent.robconf:=[0,0,0,0];
        CalcTrack:=Bed1Wyong.uframe.trans.x+pCurrent.trans.x;
        IF CurrentY<1000 THEN CalcTrack:=CalcTrack+1200; ENDIF
        IF CalcTrack<TrackMin THEN CalcTrack:=TrackMin; ENDIF
        IF CalcTrack>TrackMax THEN CalcTrack:=TrackMax; ENDIF
        pCurrent.extax:=[CalcTrack,9E+09,9E+09,9E+09,9E+09,9E+09];
        FCPressL pCurrent,v500,150,fine,tPolish\WObj:=Bed1Wyong;

        ! Work point 16: (800, 100) [work]
        CurrentX:=800;
        CurrentY:=100;
        pCurrent.trans:=[-1*CurrentX,CurrentY,WorkZ];
        pCurrent.robconf:=[0,0,0,0];
        CalcTrack:=Bed1Wyong.uframe.trans.x+pCurrent.trans.x;
        IF CurrentY<1000 THEN CalcTrack:=CalcTrack+1200; ENDIF
        IF CalcTrack<TrackMin THEN CalcTrack:=TrackMin; ENDIF
        IF CalcTrack>TrackMax THEN CalcTrack:=TrackMax; ENDIF
        pCurrent.extax:=[CalcTrack,9E+09,9E+09,9E+09,9E+09,9E+09];
        FCPressL pCurrent,v500,150,fine,tPolish\WObj:=Bed1Wyong;

        ! Work point 17: (800, 1750) [work]
        CurrentX:=800;
        CurrentY:=1750;
        pCurrent.trans:=[-1*CurrentX,CurrentY,WorkZ];
        pCurrent.robconf:=[0,0,0,0];
        CalcTrack:=Bed1Wyong.uframe.trans.x+pCurrent.trans.x;
        IF CurrentY<1000 THEN CalcTrack:=CalcTrack+1200; ENDIF
        IF CalcTrack<TrackMin THEN CalcTrack:=TrackMin; ENDIF
        IF CalcTrack>TrackMax THEN CalcTrack:=TrackMax; ENDIF
        pCurrent.extax:=[CalcTrack,9E+09,9E+09,9E+09,9E+09,9E+09];
        FCPressL pCurrent,v500,150,fine,tPolish\WObj:=Bed1Wyong;

        ! Work point 18: (1150, 1750) [work]
        CurrentX:=1150;
        CurrentY:=1750;
        pCurrent.trans:=[-1*CurrentX,CurrentY,WorkZ];
        pCurrent.robconf:=[0,0,0,0];
        CalcTrack:=Bed1Wyong.uframe.trans.x+pCurrent.trans.x;
        IF CurrentY<1000 THEN CalcTrack:=CalcTrack+1200; ENDIF
        IF CalcTrack<TrackMin THEN CalcTrack:=TrackMin; ENDIF
        IF CalcTrack>TrackMax THEN CalcTrack:=TrackMax; ENDIF
        pCurrent.extax:=[CalcTrack,9E+09,9E+09,9E+09,9E+09,9E+09];
        FCPressL pCurrent,v500,150,fine,tPolish\WObj:=Bed1Wyong;

        ! Work point 19: (1150, 100) [work]
        CurrentX:=1150;
        CurrentY:=100;
        pCurrent.trans:=[-1*CurrentX,CurrentY,WorkZ];
        pCurrent.robconf:=[0,0,0,0];
        CalcTrack:=Bed1Wyong.uframe.trans.x+pCurrent.trans.x;
        IF CurrentY<1000 THEN CalcTrack:=CalcTrack+1200; ENDIF
        IF CalcTrack<TrackMin THEN CalcTrack:=TrackMin; ENDIF
        IF CalcTrack>TrackMax THEN CalcTrack:=TrackMax; ENDIF
        pCurrent.extax:=[CalcTrack,9E+09,9E+09,9E+09,9E+09,9E+09];
        FCPressL pCurrent,v500,150,fine,tPolish\WObj:=Bed1Wyong;

        ! Work point 20: (1500, 100) [work]
        CurrentX:=1500;
        CurrentY:=100;
        pCurrent.trans:=[-1*CurrentX,CurrentY,WorkZ];
        pCurrent.robconf:=[0,0,0,0];
        CalcTrack:=Bed1Wyong.uframe.trans.x+pCurrent.trans.x;
        IF CurrentY<1000 THEN CalcTrack:=CalcTrack+1200; ENDIF
        IF CalcTrack<TrackMin THEN CalcTrack:=TrackMin; ENDIF
        IF CalcTrack>TrackMax THEN CalcTrack:=TrackMax; ENDIF
        pCurrent.extax:=[CalcTrack,9E+09,9E+09,9E+09,9E+09,9E+09];
        FCPressL pCurrent,v500,150,fine,tPolish\WObj:=Bed1Wyong;

        ! Work point 21: (1500, 1750) [work]
        CurrentX:=1500;
        CurrentY:=1750;
        pCurrent.trans:=[-1*CurrentX,CurrentY,WorkZ];
        pCurrent.robconf:=[0,0,0,0];
        CalcTrack:=Bed1Wyong.uframe.trans.x+pCurrent.trans.x;
        IF CurrentY<1000 THEN CalcTrack:=CalcTrack+1200; ENDIF
        IF CalcTrack<TrackMin THEN CalcTrack:=TrackMin; ENDIF
        IF CalcTrack>TrackMax THEN CalcTrack:=TrackMax; ENDIF
        pCurrent.extax:=[CalcTrack,9E+09,9E+09,9E+09,9E+09,9E+09];
        FCPressL pCurrent,v500,150,fine,tPolish\WObj:=Bed1Wyong;

        ! Work point 22: (1850, 1750) [work]
        CurrentX:=1850;
        CurrentY:=1750;
        pCurrent.trans:=[-1*CurrentX,CurrentY,WorkZ];
        pCurrent.robconf:=[0,0,0,0];
        CalcTrack:=Bed1Wyong.uframe.trans.x+pCurrent.trans.x;
        IF CurrentY<1000 THEN CalcTrack:=CalcTrack+1200; ENDIF
        IF CalcTrack<TrackMin THEN CalcTrack:=TrackMin; ENDIF
        IF CalcTrack>TrackMax THEN CalcTrack:=TrackMax; ENDIF
        pCurrent.extax:=[CalcTrack,9E+09,9E+09,9E+09,9E+09,9E+09];
        FCPressL pCurrent,v500,150,fine,tPolish\WObj:=Bed1Wyong;

        ! Work point 23: (1850, 100) [work]
        CurrentX:=1850;
        CurrentY:=100;
        pCurrent.trans:=[-1*CurrentX,CurrentY,WorkZ];
        pCurrent.robconf:=[0,0,0,0];
        CalcTrack:=Bed1Wyong.uframe.trans.x+pCurrent.trans.x;
        IF CurrentY<1000 THEN CalcTrack:=CalcTrack+1200; ENDIF
        IF CalcTrack<TrackMin THEN CalcTrack:=TrackMin; ENDIF
        IF CalcTrack>TrackMax THEN CalcTrack:=TrackMax; ENDIF
        pCurrent.extax:=[CalcTrack,9E+09,9E+09,9E+09,9E+09,9E+09];
        FCPressL pCurrent,v500,150,fine,tPolish\WObj:=Bed1Wyong;

        ! Work point 24: (2200, 100) [work]
        CurrentX:=2200;
        CurrentY:=100;
        pCurrent.trans:=[-1*CurrentX,CurrentY,WorkZ];
        pCurrent.robconf:=[0,0,0,0];
        CalcTrack:=Bed1Wyong.uframe.trans.x+pCurrent.trans.x;
        IF CurrentY<1000 THEN CalcTrack:=CalcTrack+1200; ENDIF
        IF CalcTrack<TrackMin THEN CalcTrack:=TrackMin; ENDIF
        IF CalcTrack>TrackMax THEN CalcTrack:=TrackMax; ENDIF
        pCurrent.extax:=[CalcTrack,9E+09,9E+09,9E+09,9E+09,9E+09];
        FCPressL pCurrent,v500,150,fine,tPolish\WObj:=Bed1Wyong;

        ! Work point 25: (2200, 1750) [work]
        CurrentX:=2200;
        CurrentY:=1750;
        pCurrent.trans:=[-1*CurrentX,CurrentY,WorkZ];
        pCurrent.robconf:=[0,0,0,0];
        CalcTrack:=Bed1Wyong.uframe.trans.x+pCurrent.trans.x;
        IF CurrentY<1000 THEN CalcTrack:=CalcTrack+1200; ENDIF
        IF CalcTrack<TrackMin THEN CalcTrack:=TrackMin; ENDIF
        IF CalcTrack>TrackMax THEN CalcTrack:=TrackMax; ENDIF
        pCurrent.extax:=[CalcTrack,9E+09,9E+09,9E+09,9E+09,9E+09];
        FCPressL pCurrent,v500,150,fine,tPolish\WObj:=Bed1Wyong;

        ! Work point 26: (2550, 1750) [work]
        CurrentX:=2550;
        CurrentY:=1750;
        pCurrent.trans:=[-1*CurrentX,CurrentY,WorkZ];
        pCurrent.robconf:=[0,0,0,0];
        CalcTrack:=Bed1Wyong.uframe.trans.x+pCurrent.trans.x;
        IF CurrentY<1000 THEN CalcTrack:=CalcTrack+1200; ENDIF
        IF CalcTrack<TrackMin THEN CalcTrack:=TrackMin; ENDIF
        IF CalcTrack>TrackMax THEN CalcTrack:=TrackMax; ENDIF
        pCurrent.extax:=[CalcTrack,9E+09,9E+09,9E+09,9E+09,9E+09];
        FCPressL pCurrent,v500,150,fine,tPolish\WObj:=Bed1Wyong;

        ! Work point 27: (2550, 100) [work]
        CurrentX:=2550;
        CurrentY:=100;
        pCurrent.trans:=[-1*CurrentX,CurrentY,WorkZ];
        pCurrent.robconf:=[0,0,0,0];
        CalcTrack:=Bed1Wyong.uframe.trans.x+pCurrent.trans.x;
        IF CurrentY<1000 THEN CalcTrack:=CalcTrack+1200; ENDIF
        IF CalcTrack<TrackMin THEN CalcTrack:=TrackMin; ENDIF
        IF CalcTrack>TrackMax THEN CalcTrack:=TrackMax; ENDIF
        pCurrent.extax:=[CalcTrack,9E+09,9E+09,9E+09,9E+09,9E+09];
        FCPressL pCurrent,v500,150,fine,tPolish\WObj:=Bed1Wyong;

        ! Work point 28: (2900, 100) [work]
        CurrentX:=2900;
        CurrentY:=100;
        pCurrent.trans:=[-1*CurrentX,CurrentY,WorkZ];
        pCurrent.robconf:=[0,0,0,0];
        CalcTrack:=Bed1Wyong.uframe.trans.x+pCurrent.trans.x;
        IF CurrentY<1000 THEN CalcTrack:=CalcTrack+1200; ENDIF
        IF CalcTrack<TrackMin THEN CalcTrack:=TrackMin; ENDIF
        IF CalcTrack>TrackMax THEN CalcTrack:=TrackMax; ENDIF
        pCurrent.extax:=[CalcTrack,9E+09,9E+09,9E+09,9E+09,9E+09];
        FCPressL pCurrent,v500,150,fine,tPolish\WObj:=Bed1Wyong;

        ! Work point 29: (2900, 1750) [work]
        CurrentX:=2900;
        CurrentY:=1750;
        pCurrent.trans:=[-1*CurrentX,CurrentY,WorkZ];
        pCurrent.robconf:=[0,0,0,0];
        CalcTrack:=Bed1Wyong.uframe.trans.x+pCurrent.trans.x;
        IF CurrentY<1000 THEN CalcTrack:=CalcTrack+1200; ENDIF
        IF CalcTrack<TrackMin THEN CalcTrack:=TrackMin; ENDIF
        IF CalcTrack>TrackMax THEN CalcTrack:=TrackMax; ENDIF
        pCurrent.extax:=[CalcTrack,9E+09,9E+09,9E+09,9E+09,9E+09];
        FCPressL pCurrent,v500,150,fine,tPolish\WObj:=Bed1Wyong;

        ! Work point 30: (3250, 1750) [work]
        CurrentX:=3250;
        CurrentY:=1750;
        pCurrent.trans:=[-1*CurrentX,CurrentY,WorkZ];
        pCurrent.robconf:=[0,0,0,0];
        CalcTrack:=Bed1Wyong.uframe.trans.x+pCurrent.trans.x;
        IF CurrentY<1000 THEN CalcTrack:=CalcTrack+1200; ENDIF
        IF CalcTrack<TrackMin THEN CalcTrack:=TrackMin; ENDIF
        IF CalcTrack>TrackMax THEN CalcTrack:=TrackMax; ENDIF
        pCurrent.extax:=[CalcTrack,9E+09,9E+09,9E+09,9E+09,9E+09];
        FCPressL pCurrent,v500,150,fine,tPolish\WObj:=Bed1Wyong;

        ! Work point 31: (3250, 100) [work]
        CurrentX:=3250;
        CurrentY:=100;
        pCurrent.trans:=[-1*CurrentX,CurrentY,WorkZ];
        pCurrent.robconf:=[0,0,0,0];
        CalcTrack:=Bed1Wyong.uframe.trans.x+pCurrent.trans.x;
        IF CurrentY<1000 THEN CalcTrack:=CalcTrack+1200; ENDIF
        IF CalcTrack<TrackMin THEN CalcTrack:=TrackMin; ENDIF
        IF CalcTrack>TrackMax THEN CalcTrack:=TrackMax; ENDIF
        pCurrent.extax:=[CalcTrack,9E+09,9E+09,9E+09,9E+09,9E+09];
        FCPressL pCurrent,v500,150,fine,tPolish\WObj:=Bed1Wyong;

        ! Work point 32: (3600, 100) [work]
        CurrentX:=3600;
        CurrentY:=100;
        pCurrent.trans:=[-1*CurrentX,CurrentY,WorkZ];
        pCurrent.robconf:=[0,0,0,0];
        CalcTrack:=Bed1Wyong.uframe.trans.x+pCurrent.trans.x;
        IF CurrentY<1000 THEN CalcTrack:=CalcTrack+1200; ENDIF
        IF CalcTrack<TrackMin THEN CalcTrack:=TrackMin; ENDIF
        IF CalcTrack>TrackMax THEN CalcTrack:=TrackMax; ENDIF
        pCurrent.extax:=[CalcTrack,9E+09,9E+09,9E+09,9E+09,9E+09];
        FCPressL pCurrent,v500,150,fine,tPolish\WObj:=Bed1Wyong;

        ! Work point 33: (3600, 1750) [work]
        CurrentX:=3600;
        CurrentY:=1750;
        pCurrent.trans:=[-1*CurrentX,CurrentY,WorkZ];
        pCurrent.robconf:=[0,0,0,0];
        CalcTrack:=Bed1Wyong.uframe.trans.x+pCurrent.trans.x;
        IF CurrentY<1000 THEN CalcTrack:=CalcTrack+1200; ENDIF
        IF CalcTrack<TrackMin THEN CalcTrack:=TrackMin; ENDIF
        IF CalcTrack>TrackMax THEN CalcTrack:=TrackMax; ENDIF
        pCurrent.extax:=[CalcTrack,9E+09,9E+09,9E+09,9E+09,9E+09];
        FCPressL pCurrent,v500,150,fine,tPolish\WObj:=Bed1Wyong;

        ! Work point 34: (3950, 1750) [work]
        CurrentX:=3950;
        CurrentY:=1750;
        pCurrent.trans:=[-1*CurrentX,CurrentY,WorkZ];
        pCurrent.robconf:=[0,0,0,0];
        CalcTrack:=Bed1Wyong.uframe.trans.x+pCurrent.trans.x;
        IF CurrentY<1000 THEN CalcTrack:=CalcTrack+1200; ENDIF
        IF CalcTrack<TrackMin THEN CalcTrack:=TrackMin; ENDIF
        IF CalcTrack>TrackMax THEN CalcTrack:=TrackMax; ENDIF
        pCurrent.extax:=[CalcTrack,9E+09,9E+09,9E+09,9E+09,9E+09];
        FCPressL pCurrent,v500,150,fine,tPolish\WObj:=Bed1Wyong;

        ! Work point 35: (3950, 100) [work]
        CurrentX:=3950;
        CurrentY:=100;
        pCurrent.trans:=[-1*CurrentX,CurrentY,WorkZ];
        pCurrent.robconf:=[0,0,0,0];
        CalcTrack:=Bed1Wyong.uframe.trans.x+pCurrent.trans.x;
        IF CurrentY<1000 THEN CalcTrack:=CalcTrack+1200; ENDIF
        IF CalcTrack<TrackMin THEN CalcTrack:=TrackMin; ENDIF
        IF CalcTrack>TrackMax THEN CalcTrack:=TrackMax; ENDIF
        pCurrent.extax:=[CalcTrack,9E+09,9E+09,9E+09,9E+09,9E+09];
        FCPressL pCurrent,v500,150,fine,tPolish\WObj:=Bed1Wyong;

        ! Work point 36: (4300, 100) [work]
        CurrentX:=4300;
        CurrentY:=100;
        pCurrent.trans:=[-1*CurrentX,CurrentY,WorkZ];
        pCurrent.robconf:=[0,0,0,0];
        CalcTrack:=Bed1Wyong.uframe.trans.x+pCurrent.trans.x;
        IF CurrentY<1000 THEN CalcTrack:=CalcTrack+1200; ENDIF
        IF CalcTrack<TrackMin THEN CalcTrack:=TrackMin; ENDIF
        IF CalcTrack>TrackMax THEN CalcTrack:=TrackMax; ENDIF
        pCurrent.extax:=[CalcTrack,9E+09,9E+09,9E+09,9E+09,9E+09];
        FCPressL pCurrent,v500,150,fine,tPolish\WObj:=Bed1Wyong;

        ! Work point 37: (4300, 1750) [work]
        CurrentX:=4300;
        CurrentY:=1750;
        pCurrent.trans:=[-1*CurrentX,CurrentY,WorkZ];
        pCurrent.robconf:=[0,0,0,0];
        CalcTrack:=Bed1Wyong.uframe.trans.x+pCurrent.trans.x;
        IF CurrentY<1000 THEN CalcTrack:=CalcTrack+1200; ENDIF
        IF CalcTrack<TrackMin THEN CalcTrack:=TrackMin; ENDIF
        IF CalcTrack>TrackMax THEN CalcTrack:=TrackMax; ENDIF
        pCurrent.extax:=[CalcTrack,9E+09,9E+09,9E+09,9E+09,9E+09];
        FCPressL pCurrent,v500,150,fine,tPolish\WObj:=Bed1Wyong;

        ! Work point 38: (4650, 1750) [work]
        CurrentX:=4650;
        CurrentY:=1750;
        pCurrent.trans:=[-1*CurrentX,CurrentY,WorkZ];
        pCurrent.robconf:=[0,0,0,0];
        CalcTrack:=Bed1Wyong.uframe.trans.x+pCurrent.trans.x;
        IF CurrentY<1000 THEN CalcTrack:=CalcTrack+1200; ENDIF
        IF CalcTrack<TrackMin THEN CalcTrack:=TrackMin; ENDIF
        IF CalcTrack>TrackMax THEN CalcTrack:=TrackMax; ENDIF
        pCurrent.extax:=[CalcTrack,9E+09,9E+09,9E+09,9E+09,9E+09];
        FCPressL pCurrent,v500,150,fine,tPolish\WObj:=Bed1Wyong;

        ! Work point 39: (4650, 100) [work]
        CurrentX:=4650;
        CurrentY:=100;
        pCurrent.trans:=[-1*CurrentX,CurrentY,WorkZ];
        pCurrent.robconf:=[0,0,0,0];
        CalcTrack:=Bed1Wyong.uframe.trans.x+pCurrent.trans.x;
        IF CurrentY<1000 THEN CalcTrack:=CalcTrack+1200; ENDIF
        IF CalcTrack<TrackMin THEN CalcTrack:=TrackMin; ENDIF
        IF CalcTrack>TrackMax THEN CalcTrack:=TrackMax; ENDIF
        pCurrent.extax:=[CalcTrack,9E+09,9E+09,9E+09,9E+09,9E+09];
        FCPressL pCurrent,v500,150,fine,tPolish\WObj:=Bed1Wyong;

        ! Work point 40: (5000, 100) [work]
        CurrentX:=5000;
        CurrentY:=100;
        pCurrent.trans:=[-1*CurrentX,CurrentY,WorkZ];
        pCurrent.robconf:=[0,0,0,0];
        CalcTrack:=Bed1Wyong.uframe.trans.x+pCurrent.trans.x;
        IF CurrentY<1000 THEN CalcTrack:=CalcTrack+1200; ENDIF
        IF CalcTrack<TrackMin THEN CalcTrack:=TrackMin; ENDIF
        IF CalcTrack>TrackMax THEN CalcTrack:=TrackMax; ENDIF
        pCurrent.extax:=[CalcTrack,9E+09,9E+09,9E+09,9E+09,9E+09];
        FCPressL pCurrent,v500,150,fine,tPolish\WObj:=Bed1Wyong;

        ! Work point 41: (5000, 1750) [work]
        CurrentX:=5000;
        CurrentY:=1750;
        pCurrent.trans:=[-1*CurrentX,CurrentY,WorkZ];
        pCurrent.robconf:=[0,0,0,0];
        CalcTrack:=Bed1Wyong.uframe.trans.x+pCurrent.trans.x;
        IF CurrentY<1000 THEN CalcTrack:=CalcTrack+1200; ENDIF
        IF CalcTrack<TrackMin THEN CalcTrack:=TrackMin; ENDIF
        IF CalcTrack>TrackMax THEN CalcTrack:=TrackMax; ENDIF
        pCurrent.extax:=[CalcTrack,9E+09,9E+09,9E+09,9E+09,9E+09];
        FCPressL pCurrent,v500,150,fine,tPolish\WObj:=Bed1Wyong;

        ! Work point 42: (5350, 1750) [work]
        CurrentX:=5350;
        CurrentY:=1750;
        pCurrent.trans:=[-1*CurrentX,CurrentY,WorkZ];
        pCurrent.robconf:=[0,0,0,0];
        CalcTrack:=Bed1Wyong.uframe.trans.x+pCurrent.trans.x;
        IF CurrentY<1000 THEN CalcTrack:=CalcTrack+1200; ENDIF
        IF CalcTrack<TrackMin THEN CalcTrack:=TrackMin; ENDIF
        IF CalcTrack>TrackMax THEN CalcTrack:=TrackMax; ENDIF
        pCurrent.extax:=[CalcTrack,9E+09,9E+09,9E+09,9E+09,9E+09];
        FCPressL pCurrent,v500,150,fine,tPolish\WObj:=Bed1Wyong;

        ! Work point 43: (5350, 100) [work]
        CurrentX:=5350;
        CurrentY:=100;
        pCurrent.trans:=[-1*CurrentX,CurrentY,WorkZ];
        pCurrent.robconf:=[0,0,0,0];
        CalcTrack:=Bed1Wyong.uframe.trans.x+pCurrent.trans.x;
        IF CurrentY<1000 THEN CalcTrack:=CalcTrack+1200; ENDIF
        IF CalcTrack<TrackMin THEN CalcTrack:=TrackMin; ENDIF
        IF CalcTrack>TrackMax THEN CalcTrack:=TrackMax; ENDIF
        pCurrent.extax:=[CalcTrack,9E+09,9E+09,9E+09,9E+09,9E+09];
        FCPressL pCurrent,v500,150,fine,tPolish\WObj:=Bed1Wyong;

        ! Work point 44: (5700, 100) [work]
        CurrentX:=5700;
        CurrentY:=100;
        pCurrent.trans:=[-1*CurrentX,CurrentY,WorkZ];
        pCurrent.robconf:=[0,0,0,0];
        CalcTrack:=Bed1Wyong.uframe.trans.x+pCurrent.trans.x;
        IF CurrentY<1000 THEN CalcTrack:=CalcTrack+1200; ENDIF
        IF CalcTrack<TrackMin THEN CalcTrack:=TrackMin; ENDIF
        IF CalcTrack>TrackMax THEN CalcTrack:=TrackMax; ENDIF
        pCurrent.extax:=[CalcTrack,9E+09,9E+09,9E+09,9E+09,9E+09];
        FCPressL pCurrent,v500,150,fine,tPolish\WObj:=Bed1Wyong;

        ! Work point 45: (5700, 1750) [work]
        CurrentX:=5700;
        CurrentY:=1750;
        pCurrent.trans:=[-1*CurrentX,CurrentY,WorkZ];
        pCurrent.robconf:=[0,0,0,0];
        CalcTrack:=Bed1Wyong.uframe.trans.x+pCurrent.trans.x;
        IF CurrentY<1000 THEN CalcTrack:=CalcTrack+1200; ENDIF
        IF CalcTrack<TrackMin THEN CalcTrack:=TrackMin; ENDIF
        IF CalcTrack>TrackMax THEN CalcTrack:=TrackMax; ENDIF
        pCurrent.extax:=[CalcTrack,9E+09,9E+09,9E+09,9E+09,9E+09];
        FCPressL pCurrent,v500,150,fine,tPolish\WObj:=Bed1Wyong;

        ! Work point 46: (6050, 1750) [work]
        CurrentX:=6050;
        CurrentY:=1750;
        pCurrent.trans:=[-1*CurrentX,CurrentY,WorkZ];
        pCurrent.robconf:=[0,0,0,0];
        CalcTrack:=Bed1Wyong.uframe.trans.x+pCurrent.trans.x;
        IF CurrentY<1000 THEN CalcTrack:=CalcTrack+1200; ENDIF
        IF CalcTrack<TrackMin THEN CalcTrack:=TrackMin; ENDIF
        IF CalcTrack>TrackMax THEN CalcTrack:=TrackMax; ENDIF
        pCurrent.extax:=[CalcTrack,9E+09,9E+09,9E+09,9E+09,9E+09];
        FCPressL pCurrent,v500,150,fine,tPolish\WObj:=Bed1Wyong;

        ! Work point 47: (6050, 100) [work]
        CurrentX:=6050;
        CurrentY:=100;
        pCurrent.trans:=[-1*CurrentX,CurrentY,WorkZ];
        pCurrent.robconf:=[0,0,0,0];
        CalcTrack:=Bed1Wyong.uframe.trans.x+pCurrent.trans.x;
        IF CurrentY<1000 THEN CalcTrack:=CalcTrack+1200; ENDIF
        IF CalcTrack<TrackMin THEN CalcTrack:=TrackMin; ENDIF
        IF CalcTrack>TrackMax THEN CalcTrack:=TrackMax; ENDIF
        pCurrent.extax:=[CalcTrack,9E+09,9E+09,9E+09,9E+09,9E+09];
        FCPressL pCurrent,v500,150,fine,tPolish\WObj:=Bed1Wyong;

        ! Work point 48: (6400, 100) [work]
        CurrentX:=6400;
        CurrentY:=100;
        pCurrent.trans:=[-1*CurrentX,CurrentY,WorkZ];
        pCurrent.robconf:=[0,0,0,0];
        CalcTrack:=Bed1Wyong.uframe.trans.x+pCurrent.trans.x;
        IF CurrentY<1000 THEN CalcTrack:=CalcTrack+1200; ENDIF
        IF CalcTrack<TrackMin THEN CalcTrack:=TrackMin; ENDIF
        IF CalcTrack>TrackMax THEN CalcTrack:=TrackMax; ENDIF
        pCurrent.extax:=[CalcTrack,9E+09,9E+09,9E+09,9E+09,9E+09];
        FCPressL pCurrent,v500,150,fine,tPolish\WObj:=Bed1Wyong;

        ! Work point 49: (6400, 1750) [work]
        CurrentX:=6400;
        CurrentY:=1750;
        pCurrent.trans:=[-1*CurrentX,CurrentY,WorkZ];
        pCurrent.robconf:=[0,0,0,0];
        CalcTrack:=Bed1Wyong.uframe.trans.x+pCurrent.trans.x;
        IF CurrentY<1000 THEN CalcTrack:=CalcTrack+1200; ENDIF
        IF CalcTrack<TrackMin THEN CalcTrack:=TrackMin; ENDIF
        IF CalcTrack>TrackMax THEN CalcTrack:=TrackMax; ENDIF
        pCurrent.extax:=[CalcTrack,9E+09,9E+09,9E+09,9E+09,9E+09];
        FCPressL pCurrent,v500,150,fine,tPolish\WObj:=Bed1Wyong;

        ! Work point 50: (6750, 1750) [work]
        CurrentX:=6750;
        CurrentY:=1750;
        pCurrent.trans:=[-1*CurrentX,CurrentY,WorkZ];
        pCurrent.robconf:=[0,0,0,0];
        CalcTrack:=Bed1Wyong.uframe.trans.x+pCurrent.trans.x;
        IF CurrentY<1000 THEN CalcTrack:=CalcTrack+1200; ENDIF
        IF CalcTrack<TrackMin THEN CalcTrack:=TrackMin; ENDIF
        IF CalcTrack>TrackMax THEN CalcTrack:=TrackMax; ENDIF
        pCurrent.extax:=[CalcTrack,9E+09,9E+09,9E+09,9E+09,9E+09];
        FCPressL pCurrent,v500,150,fine,tPolish\WObj:=Bed1Wyong;

        ! Work point 51: (6750, 100) [work]
        CurrentX:=6750;
        CurrentY:=100;
        pCurrent.trans:=[-1*CurrentX,CurrentY,WorkZ];
        pCurrent.robconf:=[0,0,0,0];
        CalcTrack:=Bed1Wyong.uframe.trans.x+pCurrent.trans.x;
        IF CurrentY<1000 THEN CalcTrack:=CalcTrack+1200; ENDIF
        IF CalcTrack<TrackMin THEN CalcTrack:=TrackMin; ENDIF
        IF CalcTrack>TrackMax THEN CalcTrack:=TrackMax; ENDIF
        pCurrent.extax:=[CalcTrack,9E+09,9E+09,9E+09,9E+09,9E+09];
        FCPressL pCurrent,v500,150,fine,tPolish\WObj:=Bed1Wyong;

        ! Work point 52: (7100, 100) [work]
        CurrentX:=7100;
        CurrentY:=100;
        pCurrent.trans:=[-1*CurrentX,CurrentY,WorkZ];
        pCurrent.robconf:=[0,0,0,0];
        CalcTrack:=Bed1Wyong.uframe.trans.x+pCurrent.trans.x;
        IF CurrentY<1000 THEN CalcTrack:=CalcTrack+1200; ENDIF
        IF CalcTrack<TrackMin THEN CalcTrack:=TrackMin; ENDIF
        IF CalcTrack>TrackMax THEN CalcTrack:=TrackMax; ENDIF
        pCurrent.extax:=[CalcTrack,9E+09,9E+09,9E+09,9E+09,9E+09];
        FCPressL pCurrent,v500,150,fine,tPolish\WObj:=Bed1Wyong;

        ! Work point 53: (7100, 1750) [work]
        CurrentX:=7100;
        CurrentY:=1750;
        pCurrent.trans:=[-1*CurrentX,CurrentY,WorkZ];
        pCurrent.robconf:=[0,0,0,0];
        CalcTrack:=Bed1Wyong.uframe.trans.x+pCurrent.trans.x;
        IF CurrentY<1000 THEN CalcTrack:=CalcTrack+1200; ENDIF
        IF CalcTrack<TrackMin THEN CalcTrack:=TrackMin; ENDIF
        IF CalcTrack>TrackMax THEN CalcTrack:=TrackMax; ENDIF
        pCurrent.extax:=[CalcTrack,9E+09,9E+09,9E+09,9E+09,9E+09];
        FCPressL pCurrent,v500,150,fine,tPolish\WObj:=Bed1Wyong;

        ! Work point 54: (7450, 1750) [work]
        CurrentX:=7450;
        CurrentY:=1750;
        pCurrent.trans:=[-1*CurrentX,CurrentY,WorkZ];
        pCurrent.robconf:=[0,0,0,0];
        CalcTrack:=Bed1Wyong.uframe.trans.x+pCurrent.trans.x;
        IF CurrentY<1000 THEN CalcTrack:=CalcTrack+1200; ENDIF
        IF CalcTrack<TrackMin THEN CalcTrack:=TrackMin; ENDIF
        IF CalcTrack>TrackMax THEN CalcTrack:=TrackMax; ENDIF
        pCurrent.extax:=[CalcTrack,9E+09,9E+09,9E+09,9E+09,9E+09];
        FCPressL pCurrent,v500,150,fine,tPolish\WObj:=Bed1Wyong;

        ! Work point 55: (7450, 100) [work]
        CurrentX:=7450;
        CurrentY:=100;
        pCurrent.trans:=[-1*CurrentX,CurrentY,WorkZ];
        pCurrent.robconf:=[0,0,0,0];
        CalcTrack:=Bed1Wyong.uframe.trans.x+pCurrent.trans.x;
        IF CurrentY<1000 THEN CalcTrack:=CalcTrack+1200; ENDIF
        IF CalcTrack<TrackMin THEN CalcTrack:=TrackMin; ENDIF
        IF CalcTrack>TrackMax THEN CalcTrack:=TrackMax; ENDIF
        pCurrent.extax:=[CalcTrack,9E+09,9E+09,9E+09,9E+09,9E+09];
        FCPressL pCurrent,v500,150,fine,tPolish\WObj:=Bed1Wyong;

        ! Work point 56: (7800, 100) [work]
        CurrentX:=7800;
        CurrentY:=100;
        pCurrent.trans:=[-1*CurrentX,CurrentY,WorkZ];
        pCurrent.robconf:=[0,0,0,0];
        CalcTrack:=Bed1Wyong.uframe.trans.x+pCurrent.trans.x;
        IF CurrentY<1000 THEN CalcTrack:=CalcTrack+1200; ENDIF
        IF CalcTrack<TrackMin THEN CalcTrack:=TrackMin; ENDIF
        IF CalcTrack>TrackMax THEN CalcTrack:=TrackMax; ENDIF
        pCurrent.extax:=[CalcTrack,9E+09,9E+09,9E+09,9E+09,9E+09];
        FCPressL pCurrent,v500,150,fine,tPolish\WObj:=Bed1Wyong;

        ! Work point 57: (7800, 1750) [work]
        CurrentX:=7800;
        CurrentY:=1750;
        pCurrent.trans:=[-1*CurrentX,CurrentY,WorkZ];
        pCurrent.robconf:=[0,0,0,0];
        CalcTrack:=Bed1Wyong.uframe.trans.x+pCurrent.trans.x;
        IF CurrentY<1000 THEN CalcTrack:=CalcTrack+1200; ENDIF
        IF CalcTrack<TrackMin THEN CalcTrack:=TrackMin; ENDIF
        IF CalcTrack>TrackMax THEN CalcTrack:=TrackMax; ENDIF
        pCurrent.extax:=[CalcTrack,9E+09,9E+09,9E+09,9E+09,9E+09];
        FCPressL pCurrent,v500,150,fine,tPolish\WObj:=Bed1Wyong;

        ! Work point 58: (8150, 1750) [work]
        CurrentX:=8150;
        CurrentY:=1750;
        pCurrent.trans:=[-1*CurrentX,CurrentY,WorkZ];
        pCurrent.robconf:=[0,0,0,0];
        CalcTrack:=Bed1Wyong.uframe.trans.x+pCurrent.trans.x;
        IF CurrentY<1000 THEN CalcTrack:=CalcTrack+1200; ENDIF
        IF CalcTrack<TrackMin THEN CalcTrack:=TrackMin; ENDIF
        IF CalcTrack>TrackMax THEN CalcTrack:=TrackMax; ENDIF
        pCurrent.extax:=[CalcTrack,9E+09,9E+09,9E+09,9E+09,9E+09];
        FCPressL pCurrent,v500,150,fine,tPolish\WObj:=Bed1Wyong;

        ! Work point 59: (8150, 100) [work]
        CurrentX:=8150;
        CurrentY:=100;
        pCurrent.trans:=[-1*CurrentX,CurrentY,WorkZ];
        pCurrent.robconf:=[0,0,0,0];
        CalcTrack:=Bed1Wyong.uframe.trans.x+pCurrent.trans.x;
        IF CurrentY<1000 THEN CalcTrack:=CalcTrack+1200; ENDIF
        IF CalcTrack<TrackMin THEN CalcTrack:=TrackMin; ENDIF
        IF CalcTrack>TrackMax THEN CalcTrack:=TrackMax; ENDIF
        pCurrent.extax:=[CalcTrack,9E+09,9E+09,9E+09,9E+09,9E+09];
        FCPressL pCurrent,v500,150,fine,tPolish\WObj:=Bed1Wyong;


        ! End force control
        CurrentJoints:=CJointT();
        CurrentPos:=CalcRobT(CurrentJoints,tPolish\WObj:=Bed1Wyong);
        FCPressEnd Offs(CurrentPos,0,0,75),v50,\DeactOnly,tPolish\WObj:=Bed1Wyong;
        bFCActive:=FALSE;

        Pol_off;

        ! Lift to safe height
        CurrentJoints:=CJointT();
        CurrentPos:=CalcRobT(CurrentJoints,tPolish\WObj:=Bed1Wyong);
        MoveL Offs(CurrentPos,0,0,200),v200,z5,tPolish\WObj:=Bed1Wyong;

        ! Return tool and go home
        TPWrite "Py2Polish: Dropping off tool...";
        Polish_Dropoff;
        Home FALSE;

        TPWrite "========================================";
        TPWrite "Py2Polish: COMPLETE";
        TPWrite "========================================";

    ERROR
        Pol_off;
        TPWrite "Py2Polish ERROR: " \Num:=ERRNO;
        RAISE;
    ENDPROC

    PROC Py2Vac()
        ! Py2Vac - Generated by Onyx Tool Class
        ! Workzone: bed
        ! Area: (200,200) to (8050,1650)
        ! Z = 295mm
        ! Step: 200mm

        VAR robtarget pCurrent;
        VAR jointtarget CurrentJoints;
        VAR robtarget CurrentPos;
        VAR num WorkZ:=295;
        VAR num SafeZ:=495;
        VAR num CurrentX:=0;
        VAR num CurrentY:=0;
        VAR speeddata vTravel:=[300,500,5000,1000];
        VAR num TrackMin:=-300;
        VAR num TrackMax:=10050;
        VAR num CalcTrack:=0;

        TPWrite "========================================";
        TPWrite "Py2Vac: Starting";
        TPWrite "========================================";
        TPWrite "Workzone: bed";
        TPWrite "WorkZ=" \Num:=WorkZ;

        ! Get tool if needed
        UpdateToolNum;
        IF ToolNum<>5 THEN
            TPWrite "Py2Vac: Getting tool...";
            Home TRUE;
            Vac_Pickup;
        ELSE
            CurrentJoints:=CJointT();
            CurrentPos:=CalcRobT(CurrentJoints,tVac\WObj:=wobj0);
            IF (CurrentPos.trans.x)>8000 AND CurrentPos.trans.z<400 THEN
                MoveL Offs(CurrentPos,0,0,(400-CurrentPos.trans.z)),v100,z5,tVac;
            ENDIF
        ENDIF

        ! Turn on vacuum
        TPWrite "Py2Vac: Starting vacuum...";
        Vac_on;
        WaitTime 1;

        ! ========================================
        ! Pattern Execution: 35 points
        ! ========================================

        ! Point 1: (200, 1650) [rapid], axis_6=180
        CurrentX:=200;
        CurrentY:=1650;
        pCurrent.trans:=[-1*CurrentX,CurrentY,SafeZ];
        pCurrent.rot:=OrientZYX(180,20,180);
        pCurrent.robconf:=[1,0,0,0];
        CalcTrack:=Bed1Wyong.uframe.trans.x+pCurrent.trans.x;
        IF CurrentY<1000 THEN CalcTrack:=CalcTrack+1200; ENDIF
        IF CalcTrack<TrackMin THEN CalcTrack:=TrackMin; ENDIF
        IF CalcTrack>TrackMax THEN CalcTrack:=TrackMax; ENDIF
        pCurrent.extax:=[CalcTrack,9E+09,9E+09,9E+09,9E+09,9E+09];
        MoveJ pCurrent,v500,z5,tVac\WObj:=Bed1Wyong;

        ! Descend to work height
        pCurrent.trans.z:=WorkZ;
        MoveL pCurrent,v100,fine,tVac\WObj:=Bed1Wyong;

        ! Point 2: (200, 1650) [work], axis_6=180
        CurrentX:=200;
        CurrentY:=1650;
        pCurrent.trans:=[-1*CurrentX,CurrentY,WorkZ];
        pCurrent.rot:=OrientZYX(180,20,180);
        pCurrent.robconf:=[1,0,0,0];
        CalcTrack:=Bed1Wyong.uframe.trans.x+pCurrent.trans.x;
        IF CurrentY<1000 THEN CalcTrack:=CalcTrack+1200; ENDIF
        IF CalcTrack<TrackMin THEN CalcTrack:=TrackMin; ENDIF
        IF CalcTrack>TrackMax THEN CalcTrack:=TrackMax; ENDIF
        pCurrent.extax:=[CalcTrack,9E+09,9E+09,9E+09,9E+09,9E+09];
        MoveL pCurrent,vTravel,fine,tVac\WObj:=Bed1Wyong;

        ! Point 3: (8050, 1650) [work], axis_6=180
        CurrentX:=8050;
        CurrentY:=1650;
        pCurrent.trans:=[-1*CurrentX,CurrentY,WorkZ];
        pCurrent.rot:=OrientZYX(180,20,180);
        pCurrent.robconf:=[1,0,0,0];
        CalcTrack:=Bed1Wyong.uframe.trans.x+pCurrent.trans.x;
        IF CurrentY<1000 THEN CalcTrack:=CalcTrack+1200; ENDIF
        IF CalcTrack<TrackMin THEN CalcTrack:=TrackMin; ENDIF
        IF CalcTrack>TrackMax THEN CalcTrack:=TrackMax; ENDIF
        pCurrent.extax:=[CalcTrack,9E+09,9E+09,9E+09,9E+09,9E+09];
        MoveL pCurrent,vTravel,fine,tVac\WObj:=Bed1Wyong;

        ! Point 4: (8050, 1450) [rapid], axis_6=180
        CurrentX:=8050;
        CurrentY:=1450;
        pCurrent.trans:=[-1*CurrentX,CurrentY,SafeZ];
        pCurrent.rot:=OrientZYX(180,20,180);
        pCurrent.robconf:=[1,0,0,0];
        CalcTrack:=Bed1Wyong.uframe.trans.x+pCurrent.trans.x;
        IF CurrentY<1000 THEN CalcTrack:=CalcTrack+1200; ENDIF
        IF CalcTrack<TrackMin THEN CalcTrack:=TrackMin; ENDIF
        IF CalcTrack>TrackMax THEN CalcTrack:=TrackMax; ENDIF
        pCurrent.extax:=[CalcTrack,9E+09,9E+09,9E+09,9E+09,9E+09];
        MoveJ pCurrent,v500,z5,tVac\WObj:=Bed1Wyong;

        ! Point 5: (8050, 1450) [rapid], axis_6=0
        CurrentX:=8050;
        CurrentY:=1450;
        pCurrent.trans:=[-1*CurrentX,CurrentY,SafeZ];
        pCurrent.rot:=OrientZYX(0,20,180);
        pCurrent.robconf:=[1,0,-2,0];
        CalcTrack:=Bed1Wyong.uframe.trans.x+pCurrent.trans.x;
        IF CurrentY<1000 THEN CalcTrack:=CalcTrack+1200; ENDIF
        IF CalcTrack<TrackMin THEN CalcTrack:=TrackMin; ENDIF
        IF CalcTrack>TrackMax THEN CalcTrack:=TrackMax; ENDIF
        pCurrent.extax:=[CalcTrack,9E+09,9E+09,9E+09,9E+09,9E+09];
        MoveJ pCurrent,v500,z5,tVac\WObj:=Bed1Wyong;

        ! Descend to work height
        pCurrent.trans.z:=WorkZ;
        MoveL pCurrent,v100,fine,tVac\WObj:=Bed1Wyong;

        ! Point 6: (8050, 1450) [work], axis_6=0
        CurrentX:=8050;
        CurrentY:=1450;
        pCurrent.trans:=[-1*CurrentX,CurrentY,WorkZ];
        pCurrent.rot:=OrientZYX(0,20,180);
        pCurrent.robconf:=[1,0,-2,0];
        CalcTrack:=Bed1Wyong.uframe.trans.x+pCurrent.trans.x;
        IF CurrentY<1000 THEN CalcTrack:=CalcTrack+1200; ENDIF
        IF CalcTrack<TrackMin THEN CalcTrack:=TrackMin; ENDIF
        IF CalcTrack>TrackMax THEN CalcTrack:=TrackMax; ENDIF
        pCurrent.extax:=[CalcTrack,9E+09,9E+09,9E+09,9E+09,9E+09];
        MoveL pCurrent,vTravel,fine,tVac\WObj:=Bed1Wyong;

        ! Point 7: (200, 1450) [work], axis_6=0
        CurrentX:=200;
        CurrentY:=1450;
        pCurrent.trans:=[-1*CurrentX,CurrentY,WorkZ];
        pCurrent.rot:=OrientZYX(0,20,180);
        pCurrent.robconf:=[1,0,-2,0];
        CalcTrack:=Bed1Wyong.uframe.trans.x+pCurrent.trans.x;
        IF CurrentY<1000 THEN CalcTrack:=CalcTrack+1200; ENDIF
        IF CalcTrack<TrackMin THEN CalcTrack:=TrackMin; ENDIF
        IF CalcTrack>TrackMax THEN CalcTrack:=TrackMax; ENDIF
        pCurrent.extax:=[CalcTrack,9E+09,9E+09,9E+09,9E+09,9E+09];
        MoveL pCurrent,vTravel,fine,tVac\WObj:=Bed1Wyong;

        ! Point 8: (200, 1250) [rapid], axis_6=0
        CurrentX:=200;
        CurrentY:=1250;
        pCurrent.trans:=[-1*CurrentX,CurrentY,SafeZ];
        pCurrent.rot:=OrientZYX(0,20,180);
        pCurrent.robconf:=[1,0,-2,0];
        CalcTrack:=Bed1Wyong.uframe.trans.x+pCurrent.trans.x;
        IF CurrentY<1000 THEN CalcTrack:=CalcTrack+1200; ENDIF
        IF CalcTrack<TrackMin THEN CalcTrack:=TrackMin; ENDIF
        IF CalcTrack>TrackMax THEN CalcTrack:=TrackMax; ENDIF
        pCurrent.extax:=[CalcTrack,9E+09,9E+09,9E+09,9E+09,9E+09];
        MoveJ pCurrent,v500,z5,tVac\WObj:=Bed1Wyong;

        ! Point 9: (200, 1250) [rapid], axis_6=180
        CurrentX:=200;
        CurrentY:=1250;
        pCurrent.trans:=[-1*CurrentX,CurrentY,SafeZ];
        pCurrent.rot:=OrientZYX(180,20,180);
        pCurrent.robconf:=[1,0,0,0];
        CalcTrack:=Bed1Wyong.uframe.trans.x+pCurrent.trans.x;
        IF CurrentY<1000 THEN CalcTrack:=CalcTrack+1200; ENDIF
        IF CalcTrack<TrackMin THEN CalcTrack:=TrackMin; ENDIF
        IF CalcTrack>TrackMax THEN CalcTrack:=TrackMax; ENDIF
        pCurrent.extax:=[CalcTrack,9E+09,9E+09,9E+09,9E+09,9E+09];
        MoveJ pCurrent,v500,z5,tVac\WObj:=Bed1Wyong;

        ! Descend to work height
        pCurrent.trans.z:=WorkZ;
        MoveL pCurrent,v100,fine,tVac\WObj:=Bed1Wyong;

        ! Point 10: (200, 1250) [work], axis_6=180
        CurrentX:=200;
        CurrentY:=1250;
        pCurrent.trans:=[-1*CurrentX,CurrentY,WorkZ];
        pCurrent.rot:=OrientZYX(180,20,180);
        pCurrent.robconf:=[1,0,0,0];
        CalcTrack:=Bed1Wyong.uframe.trans.x+pCurrent.trans.x;
        IF CurrentY<1000 THEN CalcTrack:=CalcTrack+1200; ENDIF
        IF CalcTrack<TrackMin THEN CalcTrack:=TrackMin; ENDIF
        IF CalcTrack>TrackMax THEN CalcTrack:=TrackMax; ENDIF
        pCurrent.extax:=[CalcTrack,9E+09,9E+09,9E+09,9E+09,9E+09];
        MoveL pCurrent,vTravel,fine,tVac\WObj:=Bed1Wyong;

        ! Point 11: (8050, 1250) [work], axis_6=180
        CurrentX:=8050;
        CurrentY:=1250;
        pCurrent.trans:=[-1*CurrentX,CurrentY,WorkZ];
        pCurrent.rot:=OrientZYX(180,20,180);
        pCurrent.robconf:=[1,0,0,0];
        CalcTrack:=Bed1Wyong.uframe.trans.x+pCurrent.trans.x;
        IF CurrentY<1000 THEN CalcTrack:=CalcTrack+1200; ENDIF
        IF CalcTrack<TrackMin THEN CalcTrack:=TrackMin; ENDIF
        IF CalcTrack>TrackMax THEN CalcTrack:=TrackMax; ENDIF
        pCurrent.extax:=[CalcTrack,9E+09,9E+09,9E+09,9E+09,9E+09];
        MoveL pCurrent,vTravel,fine,tVac\WObj:=Bed1Wyong;

        ! Point 12: (8050, 1050) [rapid], axis_6=180
        CurrentX:=8050;
        CurrentY:=1050;
        pCurrent.trans:=[-1*CurrentX,CurrentY,SafeZ];
        pCurrent.rot:=OrientZYX(180,20,180);
        pCurrent.robconf:=[1,0,0,0];
        CalcTrack:=Bed1Wyong.uframe.trans.x+pCurrent.trans.x;
        IF CurrentY<1000 THEN CalcTrack:=CalcTrack+1200; ENDIF
        IF CalcTrack<TrackMin THEN CalcTrack:=TrackMin; ENDIF
        IF CalcTrack>TrackMax THEN CalcTrack:=TrackMax; ENDIF
        pCurrent.extax:=[CalcTrack,9E+09,9E+09,9E+09,9E+09,9E+09];
        MoveJ pCurrent,v500,z5,tVac\WObj:=Bed1Wyong;

        ! Point 13: (8050, 1050) [rapid], axis_6=0
        CurrentX:=8050;
        CurrentY:=1050;
        pCurrent.trans:=[-1*CurrentX,CurrentY,SafeZ];
        pCurrent.rot:=OrientZYX(0,20,180);
        pCurrent.robconf:=[1,0,-2,0];
        CalcTrack:=Bed1Wyong.uframe.trans.x+pCurrent.trans.x;
        IF CurrentY<1000 THEN CalcTrack:=CalcTrack+1200; ENDIF
        IF CalcTrack<TrackMin THEN CalcTrack:=TrackMin; ENDIF
        IF CalcTrack>TrackMax THEN CalcTrack:=TrackMax; ENDIF
        pCurrent.extax:=[CalcTrack,9E+09,9E+09,9E+09,9E+09,9E+09];
        MoveJ pCurrent,v500,z5,tVac\WObj:=Bed1Wyong;

        ! Descend to work height
        pCurrent.trans.z:=WorkZ;
        MoveL pCurrent,v100,fine,tVac\WObj:=Bed1Wyong;

        ! Point 14: (8050, 1050) [work], axis_6=0
        CurrentX:=8050;
        CurrentY:=1050;
        pCurrent.trans:=[-1*CurrentX,CurrentY,WorkZ];
        pCurrent.rot:=OrientZYX(0,20,180);
        pCurrent.robconf:=[1,0,-2,0];
        CalcTrack:=Bed1Wyong.uframe.trans.x+pCurrent.trans.x;
        IF CurrentY<1000 THEN CalcTrack:=CalcTrack+1200; ENDIF
        IF CalcTrack<TrackMin THEN CalcTrack:=TrackMin; ENDIF
        IF CalcTrack>TrackMax THEN CalcTrack:=TrackMax; ENDIF
        pCurrent.extax:=[CalcTrack,9E+09,9E+09,9E+09,9E+09,9E+09];
        MoveL pCurrent,vTravel,fine,tVac\WObj:=Bed1Wyong;

        ! Point 15: (200, 1050) [work], axis_6=0
        CurrentX:=200;
        CurrentY:=1050;
        pCurrent.trans:=[-1*CurrentX,CurrentY,WorkZ];
        pCurrent.rot:=OrientZYX(0,20,180);
        pCurrent.robconf:=[1,0,-2,0];
        CalcTrack:=Bed1Wyong.uframe.trans.x+pCurrent.trans.x;
        IF CurrentY<1000 THEN CalcTrack:=CalcTrack+1200; ENDIF
        IF CalcTrack<TrackMin THEN CalcTrack:=TrackMin; ENDIF
        IF CalcTrack>TrackMax THEN CalcTrack:=TrackMax; ENDIF
        pCurrent.extax:=[CalcTrack,9E+09,9E+09,9E+09,9E+09,9E+09];
        MoveL pCurrent,vTravel,fine,tVac\WObj:=Bed1Wyong;

        ! Point 16: (200, 850) [rapid], axis_6=0
        CurrentX:=200;
        CurrentY:=850;
        pCurrent.trans:=[-1*CurrentX,CurrentY,SafeZ];
        pCurrent.rot:=OrientZYX(0,20,180);
        pCurrent.robconf:=[1,0,-2,0];
        CalcTrack:=Bed1Wyong.uframe.trans.x+pCurrent.trans.x;
        IF CurrentY<1000 THEN CalcTrack:=CalcTrack+1200; ENDIF
        IF CalcTrack<TrackMin THEN CalcTrack:=TrackMin; ENDIF
        IF CalcTrack>TrackMax THEN CalcTrack:=TrackMax; ENDIF
        pCurrent.extax:=[CalcTrack,9E+09,9E+09,9E+09,9E+09,9E+09];
        MoveJ pCurrent,v500,z5,tVac\WObj:=Bed1Wyong;

        ! Point 17: (200, 850) [rapid], axis_6=180
        CurrentX:=200;
        CurrentY:=850;
        pCurrent.trans:=[-1*CurrentX,CurrentY,SafeZ];
        pCurrent.rot:=OrientZYX(180,20,180);
        pCurrent.robconf:=[1,0,0,0];
        CalcTrack:=Bed1Wyong.uframe.trans.x+pCurrent.trans.x;
        IF CurrentY<1000 THEN CalcTrack:=CalcTrack+1200; ENDIF
        IF CalcTrack<TrackMin THEN CalcTrack:=TrackMin; ENDIF
        IF CalcTrack>TrackMax THEN CalcTrack:=TrackMax; ENDIF
        pCurrent.extax:=[CalcTrack,9E+09,9E+09,9E+09,9E+09,9E+09];
        MoveJ pCurrent,v500,z5,tVac\WObj:=Bed1Wyong;

        ! Descend to work height
        pCurrent.trans.z:=WorkZ;
        MoveL pCurrent,v100,fine,tVac\WObj:=Bed1Wyong;

        ! Point 18: (200, 850) [work], axis_6=180
        CurrentX:=200;
        CurrentY:=850;
        pCurrent.trans:=[-1*CurrentX,CurrentY,WorkZ];
        pCurrent.rot:=OrientZYX(180,20,180);
        pCurrent.robconf:=[1,0,0,0];
        CalcTrack:=Bed1Wyong.uframe.trans.x+pCurrent.trans.x;
        IF CurrentY<1000 THEN CalcTrack:=CalcTrack+1200; ENDIF
        IF CalcTrack<TrackMin THEN CalcTrack:=TrackMin; ENDIF
        IF CalcTrack>TrackMax THEN CalcTrack:=TrackMax; ENDIF
        pCurrent.extax:=[CalcTrack,9E+09,9E+09,9E+09,9E+09,9E+09];
        MoveL pCurrent,vTravel,fine,tVac\WObj:=Bed1Wyong;

        ! Point 19: (8050, 850) [work], axis_6=180
        CurrentX:=8050;
        CurrentY:=850;
        pCurrent.trans:=[-1*CurrentX,CurrentY,WorkZ];
        pCurrent.rot:=OrientZYX(180,20,180);
        pCurrent.robconf:=[1,0,0,0];
        CalcTrack:=Bed1Wyong.uframe.trans.x+pCurrent.trans.x;
        IF CurrentY<1000 THEN CalcTrack:=CalcTrack+1200; ENDIF
        IF CalcTrack<TrackMin THEN CalcTrack:=TrackMin; ENDIF
        IF CalcTrack>TrackMax THEN CalcTrack:=TrackMax; ENDIF
        pCurrent.extax:=[CalcTrack,9E+09,9E+09,9E+09,9E+09,9E+09];
        MoveL pCurrent,vTravel,fine,tVac\WObj:=Bed1Wyong;

        ! Point 20: (8050, 650) [rapid], axis_6=180
        CurrentX:=8050;
        CurrentY:=650;
        pCurrent.trans:=[-1*CurrentX,CurrentY,SafeZ];
        pCurrent.rot:=OrientZYX(180,20,180);
        pCurrent.robconf:=[1,0,0,0];
        CalcTrack:=Bed1Wyong.uframe.trans.x+pCurrent.trans.x;
        IF CurrentY<1000 THEN CalcTrack:=CalcTrack+1200; ENDIF
        IF CalcTrack<TrackMin THEN CalcTrack:=TrackMin; ENDIF
        IF CalcTrack>TrackMax THEN CalcTrack:=TrackMax; ENDIF
        pCurrent.extax:=[CalcTrack,9E+09,9E+09,9E+09,9E+09,9E+09];
        MoveJ pCurrent,v500,z5,tVac\WObj:=Bed1Wyong;

        ! Point 21: (8050, 650) [rapid], axis_6=0
        CurrentX:=8050;
        CurrentY:=650;
        pCurrent.trans:=[-1*CurrentX,CurrentY,SafeZ];
        pCurrent.rot:=OrientZYX(0,20,180);
        pCurrent.robconf:=[1,0,-2,0];
        CalcTrack:=Bed1Wyong.uframe.trans.x+pCurrent.trans.x;
        IF CurrentY<1000 THEN CalcTrack:=CalcTrack+1200; ENDIF
        IF CalcTrack<TrackMin THEN CalcTrack:=TrackMin; ENDIF
        IF CalcTrack>TrackMax THEN CalcTrack:=TrackMax; ENDIF
        pCurrent.extax:=[CalcTrack,9E+09,9E+09,9E+09,9E+09,9E+09];
        MoveJ pCurrent,v500,z5,tVac\WObj:=Bed1Wyong;

        ! Descend to work height
        pCurrent.trans.z:=WorkZ;
        MoveL pCurrent,v100,fine,tVac\WObj:=Bed1Wyong;

        ! Point 22: (8050, 650) [work], axis_6=0
        CurrentX:=8050;
        CurrentY:=650;
        pCurrent.trans:=[-1*CurrentX,CurrentY,WorkZ];
        pCurrent.rot:=OrientZYX(0,20,180);
        pCurrent.robconf:=[1,0,-2,0];
        CalcTrack:=Bed1Wyong.uframe.trans.x+pCurrent.trans.x;
        IF CurrentY<1000 THEN CalcTrack:=CalcTrack+1200; ENDIF
        IF CalcTrack<TrackMin THEN CalcTrack:=TrackMin; ENDIF
        IF CalcTrack>TrackMax THEN CalcTrack:=TrackMax; ENDIF
        pCurrent.extax:=[CalcTrack,9E+09,9E+09,9E+09,9E+09,9E+09];
        MoveL pCurrent,vTravel,fine,tVac\WObj:=Bed1Wyong;

        ! Point 23: (200, 650) [work], axis_6=0
        CurrentX:=200;
        CurrentY:=650;
        pCurrent.trans:=[-1*CurrentX,CurrentY,WorkZ];
        pCurrent.rot:=OrientZYX(0,20,180);
        pCurrent.robconf:=[1,0,-2,0];
        CalcTrack:=Bed1Wyong.uframe.trans.x+pCurrent.trans.x;
        IF CurrentY<1000 THEN CalcTrack:=CalcTrack+1200; ENDIF
        IF CalcTrack<TrackMin THEN CalcTrack:=TrackMin; ENDIF
        IF CalcTrack>TrackMax THEN CalcTrack:=TrackMax; ENDIF
        pCurrent.extax:=[CalcTrack,9E+09,9E+09,9E+09,9E+09,9E+09];
        MoveL pCurrent,vTravel,fine,tVac\WObj:=Bed1Wyong;

        ! Point 24: (200, 450) [rapid], axis_6=0
        CurrentX:=200;
        CurrentY:=450;
        pCurrent.trans:=[-1*CurrentX,CurrentY,SafeZ];
        pCurrent.rot:=OrientZYX(0,20,180);
        pCurrent.robconf:=[1,0,-2,0];
        CalcTrack:=Bed1Wyong.uframe.trans.x+pCurrent.trans.x;
        IF CurrentY<1000 THEN CalcTrack:=CalcTrack+1200; ENDIF
        IF CalcTrack<TrackMin THEN CalcTrack:=TrackMin; ENDIF
        IF CalcTrack>TrackMax THEN CalcTrack:=TrackMax; ENDIF
        pCurrent.extax:=[CalcTrack,9E+09,9E+09,9E+09,9E+09,9E+09];
        MoveJ pCurrent,v500,z5,tVac\WObj:=Bed1Wyong;

        ! Point 25: (200, 450) [rapid], axis_6=180
        CurrentX:=200;
        CurrentY:=450;
        pCurrent.trans:=[-1*CurrentX,CurrentY,SafeZ];
        pCurrent.rot:=OrientZYX(180,20,180);
        pCurrent.robconf:=[1,0,0,0];
        CalcTrack:=Bed1Wyong.uframe.trans.x+pCurrent.trans.x;
        IF CurrentY<1000 THEN CalcTrack:=CalcTrack+1200; ENDIF
        IF CalcTrack<TrackMin THEN CalcTrack:=TrackMin; ENDIF
        IF CalcTrack>TrackMax THEN CalcTrack:=TrackMax; ENDIF
        pCurrent.extax:=[CalcTrack,9E+09,9E+09,9E+09,9E+09,9E+09];
        MoveJ pCurrent,v500,z5,tVac\WObj:=Bed1Wyong;

        ! Descend to work height
        pCurrent.trans.z:=WorkZ;
        MoveL pCurrent,v100,fine,tVac\WObj:=Bed1Wyong;

        ! Point 26: (200, 450) [work], axis_6=180
        CurrentX:=200;
        CurrentY:=450;
        pCurrent.trans:=[-1*CurrentX,CurrentY,WorkZ];
        pCurrent.rot:=OrientZYX(180,20,180);
        pCurrent.robconf:=[1,0,0,0];
        CalcTrack:=Bed1Wyong.uframe.trans.x+pCurrent.trans.x;
        IF CurrentY<1000 THEN CalcTrack:=CalcTrack+1200; ENDIF
        IF CalcTrack<TrackMin THEN CalcTrack:=TrackMin; ENDIF
        IF CalcTrack>TrackMax THEN CalcTrack:=TrackMax; ENDIF
        pCurrent.extax:=[CalcTrack,9E+09,9E+09,9E+09,9E+09,9E+09];
        MoveL pCurrent,vTravel,fine,tVac\WObj:=Bed1Wyong;

        ! Point 27: (8050, 450) [work], axis_6=180
        CurrentX:=8050;
        CurrentY:=450;
        pCurrent.trans:=[-1*CurrentX,CurrentY,WorkZ];
        pCurrent.rot:=OrientZYX(180,20,180);
        pCurrent.robconf:=[1,0,0,0];
        CalcTrack:=Bed1Wyong.uframe.trans.x+pCurrent.trans.x;
        IF CurrentY<1000 THEN CalcTrack:=CalcTrack+1200; ENDIF
        IF CalcTrack<TrackMin THEN CalcTrack:=TrackMin; ENDIF
        IF CalcTrack>TrackMax THEN CalcTrack:=TrackMax; ENDIF
        pCurrent.extax:=[CalcTrack,9E+09,9E+09,9E+09,9E+09,9E+09];
        MoveL pCurrent,vTravel,fine,tVac\WObj:=Bed1Wyong;

        ! Point 28: (8050, 250) [rapid], axis_6=180
        CurrentX:=8050;
        CurrentY:=250;
        pCurrent.trans:=[-1*CurrentX,CurrentY,SafeZ];
        pCurrent.rot:=OrientZYX(180,20,180);
        pCurrent.robconf:=[1,0,0,0];
        CalcTrack:=Bed1Wyong.uframe.trans.x+pCurrent.trans.x;
        IF CurrentY<1000 THEN CalcTrack:=CalcTrack+1200; ENDIF
        IF CalcTrack<TrackMin THEN CalcTrack:=TrackMin; ENDIF
        IF CalcTrack>TrackMax THEN CalcTrack:=TrackMax; ENDIF
        pCurrent.extax:=[CalcTrack,9E+09,9E+09,9E+09,9E+09,9E+09];
        MoveJ pCurrent,v500,z5,tVac\WObj:=Bed1Wyong;

        ! Point 29: (8050, 250) [rapid], axis_6=0
        CurrentX:=8050;
        CurrentY:=250;
        pCurrent.trans:=[-1*CurrentX,CurrentY,SafeZ];
        pCurrent.rot:=OrientZYX(0,20,180);
        pCurrent.robconf:=[1,0,-2,0];
        CalcTrack:=Bed1Wyong.uframe.trans.x+pCurrent.trans.x;
        IF CurrentY<1000 THEN CalcTrack:=CalcTrack+1200; ENDIF
        IF CalcTrack<TrackMin THEN CalcTrack:=TrackMin; ENDIF
        IF CalcTrack>TrackMax THEN CalcTrack:=TrackMax; ENDIF
        pCurrent.extax:=[CalcTrack,9E+09,9E+09,9E+09,9E+09,9E+09];
        MoveJ pCurrent,v500,z5,tVac\WObj:=Bed1Wyong;

        ! Descend to work height
        pCurrent.trans.z:=WorkZ;
        MoveL pCurrent,v100,fine,tVac\WObj:=Bed1Wyong;

        ! Point 30: (8050, 250) [work], axis_6=0
        CurrentX:=8050;
        CurrentY:=250;
        pCurrent.trans:=[-1*CurrentX,CurrentY,WorkZ];
        pCurrent.rot:=OrientZYX(0,20,180);
        pCurrent.robconf:=[1,0,-2,0];
        CalcTrack:=Bed1Wyong.uframe.trans.x+pCurrent.trans.x;
        IF CurrentY<1000 THEN CalcTrack:=CalcTrack+1200; ENDIF
        IF CalcTrack<TrackMin THEN CalcTrack:=TrackMin; ENDIF
        IF CalcTrack>TrackMax THEN CalcTrack:=TrackMax; ENDIF
        pCurrent.extax:=[CalcTrack,9E+09,9E+09,9E+09,9E+09,9E+09];
        MoveL pCurrent,vTravel,fine,tVac\WObj:=Bed1Wyong;

        ! Point 31: (200, 250) [work], axis_6=0
        CurrentX:=200;
        CurrentY:=250;
        pCurrent.trans:=[-1*CurrentX,CurrentY,WorkZ];
        pCurrent.rot:=OrientZYX(0,20,180);
        pCurrent.robconf:=[1,0,-2,0];
        CalcTrack:=Bed1Wyong.uframe.trans.x+pCurrent.trans.x;
        IF CurrentY<1000 THEN CalcTrack:=CalcTrack+1200; ENDIF
        IF CalcTrack<TrackMin THEN CalcTrack:=TrackMin; ENDIF
        IF CalcTrack>TrackMax THEN CalcTrack:=TrackMax; ENDIF
        pCurrent.extax:=[CalcTrack,9E+09,9E+09,9E+09,9E+09,9E+09];
        MoveL pCurrent,vTravel,fine,tVac\WObj:=Bed1Wyong;

        ! Point 32: (200, 200) [rapid], axis_6=0
        CurrentX:=200;
        CurrentY:=200;
        pCurrent.trans:=[-1*CurrentX,CurrentY,SafeZ];
        pCurrent.rot:=OrientZYX(0,20,180);
        pCurrent.robconf:=[1,0,-2,0];
        CalcTrack:=Bed1Wyong.uframe.trans.x+pCurrent.trans.x;
        IF CurrentY<1000 THEN CalcTrack:=CalcTrack+1200; ENDIF
        IF CalcTrack<TrackMin THEN CalcTrack:=TrackMin; ENDIF
        IF CalcTrack>TrackMax THEN CalcTrack:=TrackMax; ENDIF
        pCurrent.extax:=[CalcTrack,9E+09,9E+09,9E+09,9E+09,9E+09];
        MoveJ pCurrent,v500,z5,tVac\WObj:=Bed1Wyong;

        ! Point 33: (200, 200) [rapid], axis_6=180
        CurrentX:=200;
        CurrentY:=200;
        pCurrent.trans:=[-1*CurrentX,CurrentY,SafeZ];
        pCurrent.rot:=OrientZYX(180,20,180);
        pCurrent.robconf:=[1,0,0,0];
        CalcTrack:=Bed1Wyong.uframe.trans.x+pCurrent.trans.x;
        IF CurrentY<1000 THEN CalcTrack:=CalcTrack+1200; ENDIF
        IF CalcTrack<TrackMin THEN CalcTrack:=TrackMin; ENDIF
        IF CalcTrack>TrackMax THEN CalcTrack:=TrackMax; ENDIF
        pCurrent.extax:=[CalcTrack,9E+09,9E+09,9E+09,9E+09,9E+09];
        MoveJ pCurrent,v500,z5,tVac\WObj:=Bed1Wyong;

        ! Descend to work height
        pCurrent.trans.z:=WorkZ;
        MoveL pCurrent,v100,fine,tVac\WObj:=Bed1Wyong;

        ! Point 34: (200, 200) [work], axis_6=180
        CurrentX:=200;
        CurrentY:=200;
        pCurrent.trans:=[-1*CurrentX,CurrentY,WorkZ];
        pCurrent.rot:=OrientZYX(180,20,180);
        pCurrent.robconf:=[1,0,0,0];
        CalcTrack:=Bed1Wyong.uframe.trans.x+pCurrent.trans.x;
        IF CurrentY<1000 THEN CalcTrack:=CalcTrack+1200; ENDIF
        IF CalcTrack<TrackMin THEN CalcTrack:=TrackMin; ENDIF
        IF CalcTrack>TrackMax THEN CalcTrack:=TrackMax; ENDIF
        pCurrent.extax:=[CalcTrack,9E+09,9E+09,9E+09,9E+09,9E+09];
        MoveL pCurrent,vTravel,fine,tVac\WObj:=Bed1Wyong;

        ! Point 35: (8050, 200) [work], axis_6=180
        CurrentX:=8050;
        CurrentY:=200;
        pCurrent.trans:=[-1*CurrentX,CurrentY,WorkZ];
        pCurrent.rot:=OrientZYX(180,20,180);
        pCurrent.robconf:=[1,0,0,0];
        CalcTrack:=Bed1Wyong.uframe.trans.x+pCurrent.trans.x;
        IF CurrentY<1000 THEN CalcTrack:=CalcTrack+1200; ENDIF
        IF CalcTrack<TrackMin THEN CalcTrack:=TrackMin; ENDIF
        IF CalcTrack>TrackMax THEN CalcTrack:=TrackMax; ENDIF
        pCurrent.extax:=[CalcTrack,9E+09,9E+09,9E+09,9E+09,9E+09];
        MoveL pCurrent,vTravel,fine,tVac\WObj:=Bed1Wyong;

        Vac_off;

        ! Lift to safe height
        CurrentJoints:=CJointT();
        CurrentPos:=CalcRobT(CurrentJoints,tVac\WObj:=Bed1Wyong);
        MoveL Offs(CurrentPos,0,0,200),v200,z5,tVac\WObj:=Bed1Wyong;

        ! Return tool and go home
        TPWrite "Py2Vac: Dropping off tool...";
        Vac_Dropoff;
        Home FALSE;

        TPWrite "========================================";
        TPWrite "Py2Vac: COMPLETE";
        TPWrite "========================================";

    ERROR
        Vac_off;
        TPWrite "Py2Vac ERROR: " \Num:=ERRNO;
        RAISE;
    ENDPROC

    PROC Py2Pan()
        ! Py2Pan - Generated by Onyx Tool Class
        ! Workzone: panel
        ! Area: (530,300) to (5930,1550)
        ! Z = 456mm
        ! Step: 300mm

        VAR robtarget pCurrent;
        VAR jointtarget CurrentJoints;
        VAR robtarget CurrentPos;
        VAR num WorkZ:=456;
        VAR num SafeZ:=656;
        VAR num CurrentX:=0;
        VAR num CurrentY:=0;
        VAR speeddata vTravel:=[100,500,5000,1000];
        VAR num TrackMin:=-300;
        VAR num TrackMax:=10050;
        VAR num CalcTrack:=0;
        VAR num PanForce:=0;
        VAR bool bFCActive:=FALSE;

        TPWrite "========================================";
        TPWrite "Py2Pan: Starting";
        TPWrite "========================================";
        TPWrite "Workzone: panel";
        TPWrite "WorkZ=" \Num:=WorkZ;

        ! Get helicopter tool (Pan attaches to it)
        UpdateToolNum;
        IF ToolNum<>2 THEN
            TPWrite "Py2Pan: Getting helicopter...";
            Home TRUE;
            Heli_Pickup;
        ELSE
            CurrentJoints:=CJointT();
            CurrentPos:=CalcRobT(CurrentJoints,tHeli\WObj:=wobj0);
            IF (CurrentPos.trans.x)>8000 AND CurrentPos.trans.z<400 THEN
                MoveL Offs(CurrentPos,0,0,(400-CurrentPos.trans.z)),v100,z5,tHeli;
            ENDIF
        ENDIF

        ! Set blade angle = 0 for pan
        HeliBlade_Angle 0;

        ! ========================================
        ! Pattern Execution: 50 points
        ! ========================================

        ! Point 1: (530, 1550) [rapid]
        CurrentX:=530;
        CurrentY:=1550;
        pCurrent.trans:=[-1*CurrentX,CurrentY,SafeZ];
        pCurrent.rot:=OrientZYX(0,0,180);
        pCurrent.robconf:=[1,0,-2,0];
        CalcTrack:=Bed1Wyong.uframe.trans.x+pCurrent.trans.x;
        IF CurrentY<1000 THEN CalcTrack:=CalcTrack+1200; ENDIF
        IF CalcTrack<TrackMin THEN CalcTrack:=TrackMin; ENDIF
        IF CalcTrack>TrackMax THEN CalcTrack:=TrackMax; ENDIF
        pCurrent.extax:=[CalcTrack,9E+09,9E+09,9E+09,9E+09,9E+09];
        MoveJ pCurrent,v500,z5,tHeli\WObj:=Bed1Wyong;

        ! Descend to work height
        pCurrent.trans.z:=WorkZ;
        MoveL pCurrent,v100,fine,tHeli\WObj:=Bed1Wyong;

        ! Point 2: (5930, 1550) [work]
        CurrentX:=5930;
        CurrentY:=1550;
        pCurrent.trans:=[-1*CurrentX,CurrentY,WorkZ];
        pCurrent.rot:=OrientZYX(0,0,180);
        pCurrent.robconf:=[1,0,-2,0];
        CalcTrack:=Bed1Wyong.uframe.trans.x+pCurrent.trans.x;
        IF CurrentY<1000 THEN CalcTrack:=CalcTrack+1200; ENDIF
        IF CalcTrack<TrackMin THEN CalcTrack:=TrackMin; ENDIF
        IF CalcTrack>TrackMax THEN CalcTrack:=TrackMax; ENDIF
        pCurrent.extax:=[CalcTrack,9E+09,9E+09,9E+09,9E+09,9E+09];
        MoveL pCurrent,vTravel,fine,tHeli\WObj:=Bed1Wyong;

        ! Point 3: (5930, 1250) [work]
        CurrentX:=5930;
        CurrentY:=1250;
        pCurrent.trans:=[-1*CurrentX,CurrentY,WorkZ];
        pCurrent.rot:=OrientZYX(0,0,180);
        pCurrent.robconf:=[1,0,-2,0];
        CalcTrack:=Bed1Wyong.uframe.trans.x+pCurrent.trans.x;
        IF CurrentY<1000 THEN CalcTrack:=CalcTrack+1200; ENDIF
        IF CalcTrack<TrackMin THEN CalcTrack:=TrackMin; ENDIF
        IF CalcTrack>TrackMax THEN CalcTrack:=TrackMax; ENDIF
        pCurrent.extax:=[CalcTrack,9E+09,9E+09,9E+09,9E+09,9E+09];
        MoveL pCurrent,vTravel,fine,tHeli\WObj:=Bed1Wyong;

        ! Point 4: (530, 1250) [work]
        CurrentX:=530;
        CurrentY:=1250;
        pCurrent.trans:=[-1*CurrentX,CurrentY,WorkZ];
        pCurrent.rot:=OrientZYX(0,0,180);
        pCurrent.robconf:=[1,0,-2,0];
        CalcTrack:=Bed1Wyong.uframe.trans.x+pCurrent.trans.x;
        IF CurrentY<1000 THEN CalcTrack:=CalcTrack+1200; ENDIF
        IF CalcTrack<TrackMin THEN CalcTrack:=TrackMin; ENDIF
        IF CalcTrack>TrackMax THEN CalcTrack:=TrackMax; ENDIF
        pCurrent.extax:=[CalcTrack,9E+09,9E+09,9E+09,9E+09,9E+09];
        MoveL pCurrent,vTravel,fine,tHeli\WObj:=Bed1Wyong;

        ! Point 5: (530, 950) [work]
        CurrentX:=530;
        CurrentY:=950;
        pCurrent.trans:=[-1*CurrentX,CurrentY,WorkZ];
        pCurrent.rot:=OrientZYX(0,0,180);
        pCurrent.robconf:=[1,0,-2,0];
        CalcTrack:=Bed1Wyong.uframe.trans.x+pCurrent.trans.x;
        IF CurrentY<1000 THEN CalcTrack:=CalcTrack+1200; ENDIF
        IF CalcTrack<TrackMin THEN CalcTrack:=TrackMin; ENDIF
        IF CalcTrack>TrackMax THEN CalcTrack:=TrackMax; ENDIF
        pCurrent.extax:=[CalcTrack,9E+09,9E+09,9E+09,9E+09,9E+09];
        MoveL pCurrent,vTravel,fine,tHeli\WObj:=Bed1Wyong;

        ! Point 6: (5930, 950) [work]
        CurrentX:=5930;
        CurrentY:=950;
        pCurrent.trans:=[-1*CurrentX,CurrentY,WorkZ];
        pCurrent.rot:=OrientZYX(0,0,180);
        pCurrent.robconf:=[1,0,-2,0];
        CalcTrack:=Bed1Wyong.uframe.trans.x+pCurrent.trans.x;
        IF CurrentY<1000 THEN CalcTrack:=CalcTrack+1200; ENDIF
        IF CalcTrack<TrackMin THEN CalcTrack:=TrackMin; ENDIF
        IF CalcTrack>TrackMax THEN CalcTrack:=TrackMax; ENDIF
        pCurrent.extax:=[CalcTrack,9E+09,9E+09,9E+09,9E+09,9E+09];
        MoveL pCurrent,vTravel,fine,tHeli\WObj:=Bed1Wyong;

        ! Point 7: (5930, 650) [work]
        CurrentX:=5930;
        CurrentY:=650;
        pCurrent.trans:=[-1*CurrentX,CurrentY,WorkZ];
        pCurrent.rot:=OrientZYX(0,0,180);
        pCurrent.robconf:=[1,0,-2,0];
        CalcTrack:=Bed1Wyong.uframe.trans.x+pCurrent.trans.x;
        IF CurrentY<1000 THEN CalcTrack:=CalcTrack+1200; ENDIF
        IF CalcTrack<TrackMin THEN CalcTrack:=TrackMin; ENDIF
        IF CalcTrack>TrackMax THEN CalcTrack:=TrackMax; ENDIF
        pCurrent.extax:=[CalcTrack,9E+09,9E+09,9E+09,9E+09,9E+09];
        MoveL pCurrent,vTravel,fine,tHeli\WObj:=Bed1Wyong;

        ! Point 8: (530, 650) [work]
        CurrentX:=530;
        CurrentY:=650;
        pCurrent.trans:=[-1*CurrentX,CurrentY,WorkZ];
        pCurrent.rot:=OrientZYX(0,0,180);
        pCurrent.robconf:=[1,0,-2,0];
        CalcTrack:=Bed1Wyong.uframe.trans.x+pCurrent.trans.x;
        IF CurrentY<1000 THEN CalcTrack:=CalcTrack+1200; ENDIF
        IF CalcTrack<TrackMin THEN CalcTrack:=TrackMin; ENDIF
        IF CalcTrack>TrackMax THEN CalcTrack:=TrackMax; ENDIF
        pCurrent.extax:=[CalcTrack,9E+09,9E+09,9E+09,9E+09,9E+09];
        MoveL pCurrent,vTravel,fine,tHeli\WObj:=Bed1Wyong;

        ! Point 9: (530, 350) [work]
        CurrentX:=530;
        CurrentY:=350;
        pCurrent.trans:=[-1*CurrentX,CurrentY,WorkZ];
        pCurrent.rot:=OrientZYX(0,0,180);
        pCurrent.robconf:=[1,0,-2,0];
        CalcTrack:=Bed1Wyong.uframe.trans.x+pCurrent.trans.x;
        IF CurrentY<1000 THEN CalcTrack:=CalcTrack+1200; ENDIF
        IF CalcTrack<TrackMin THEN CalcTrack:=TrackMin; ENDIF
        IF CalcTrack>TrackMax THEN CalcTrack:=TrackMax; ENDIF
        pCurrent.extax:=[CalcTrack,9E+09,9E+09,9E+09,9E+09,9E+09];
        MoveL pCurrent,vTravel,fine,tHeli\WObj:=Bed1Wyong;

        ! Point 10: (5930, 350) [work]
        CurrentX:=5930;
        CurrentY:=350;
        pCurrent.trans:=[-1*CurrentX,CurrentY,WorkZ];
        pCurrent.rot:=OrientZYX(0,0,180);
        pCurrent.robconf:=[1,0,-2,0];
        CalcTrack:=Bed1Wyong.uframe.trans.x+pCurrent.trans.x;
        IF CurrentY<1000 THEN CalcTrack:=CalcTrack+1200; ENDIF
        IF CalcTrack<TrackMin THEN CalcTrack:=TrackMin; ENDIF
        IF CalcTrack>TrackMax THEN CalcTrack:=TrackMax; ENDIF
        pCurrent.extax:=[CalcTrack,9E+09,9E+09,9E+09,9E+09,9E+09];
        MoveL pCurrent,vTravel,fine,tHeli\WObj:=Bed1Wyong;

        ! Point 11: (5930, 300) [work]
        CurrentX:=5930;
        CurrentY:=300;
        pCurrent.trans:=[-1*CurrentX,CurrentY,WorkZ];
        pCurrent.rot:=OrientZYX(0,0,180);
        pCurrent.robconf:=[1,0,-2,0];
        CalcTrack:=Bed1Wyong.uframe.trans.x+pCurrent.trans.x;
        IF CurrentY<1000 THEN CalcTrack:=CalcTrack+1200; ENDIF
        IF CalcTrack<TrackMin THEN CalcTrack:=TrackMin; ENDIF
        IF CalcTrack>TrackMax THEN CalcTrack:=TrackMax; ENDIF
        pCurrent.extax:=[CalcTrack,9E+09,9E+09,9E+09,9E+09,9E+09];
        MoveL pCurrent,vTravel,fine,tHeli\WObj:=Bed1Wyong;

        ! Point 12: (530, 300) [work]
        CurrentX:=530;
        CurrentY:=300;
        pCurrent.trans:=[-1*CurrentX,CurrentY,WorkZ];
        pCurrent.rot:=OrientZYX(0,0,180);
        pCurrent.robconf:=[1,0,-2,0];
        CalcTrack:=Bed1Wyong.uframe.trans.x+pCurrent.trans.x;
        IF CurrentY<1000 THEN CalcTrack:=CalcTrack+1200; ENDIF
        IF CalcTrack<TrackMin THEN CalcTrack:=TrackMin; ENDIF
        IF CalcTrack>TrackMax THEN CalcTrack:=TrackMax; ENDIF
        pCurrent.extax:=[CalcTrack,9E+09,9E+09,9E+09,9E+09,9E+09];
        MoveL pCurrent,vTravel,fine,tHeli\WObj:=Bed1Wyong;

        ! Point 13: (530, 300) [work]
        CurrentX:=530;
        CurrentY:=300;
        pCurrent.trans:=[-1*CurrentX,CurrentY,WorkZ];
        pCurrent.rot:=OrientZYX(0,0,180);
        pCurrent.robconf:=[1,0,-2,0];
        CalcTrack:=Bed1Wyong.uframe.trans.x+pCurrent.trans.x;
        IF CurrentY<1000 THEN CalcTrack:=CalcTrack+1200; ENDIF
        IF CalcTrack<TrackMin THEN CalcTrack:=TrackMin; ENDIF
        IF CalcTrack>TrackMax THEN CalcTrack:=TrackMax; ENDIF
        pCurrent.extax:=[CalcTrack,9E+09,9E+09,9E+09,9E+09,9E+09];
        MoveL pCurrent,vTravel,fine,tHeli\WObj:=Bed1Wyong;

        ! Point 14: (530, 1550) [work]
        CurrentX:=530;
        CurrentY:=1550;
        pCurrent.trans:=[-1*CurrentX,CurrentY,WorkZ];
        pCurrent.rot:=OrientZYX(0,0,180);
        pCurrent.robconf:=[1,0,-2,0];
        CalcTrack:=Bed1Wyong.uframe.trans.x+pCurrent.trans.x;
        IF CurrentY<1000 THEN CalcTrack:=CalcTrack+1200; ENDIF
        IF CalcTrack<TrackMin THEN CalcTrack:=TrackMin; ENDIF
        IF CalcTrack>TrackMax THEN CalcTrack:=TrackMax; ENDIF
        pCurrent.extax:=[CalcTrack,9E+09,9E+09,9E+09,9E+09,9E+09];
        MoveL pCurrent,vTravel,fine,tHeli\WObj:=Bed1Wyong;

        ! Point 15: (830, 1550) [work]
        CurrentX:=830;
        CurrentY:=1550;
        pCurrent.trans:=[-1*CurrentX,CurrentY,WorkZ];
        pCurrent.rot:=OrientZYX(0,0,180);
        pCurrent.robconf:=[1,0,-2,0];
        CalcTrack:=Bed1Wyong.uframe.trans.x+pCurrent.trans.x;
        IF CurrentY<1000 THEN CalcTrack:=CalcTrack+1200; ENDIF
        IF CalcTrack<TrackMin THEN CalcTrack:=TrackMin; ENDIF
        IF CalcTrack>TrackMax THEN CalcTrack:=TrackMax; ENDIF
        pCurrent.extax:=[CalcTrack,9E+09,9E+09,9E+09,9E+09,9E+09];
        MoveL pCurrent,vTravel,fine,tHeli\WObj:=Bed1Wyong;

        ! Point 16: (830, 300) [work]
        CurrentX:=830;
        CurrentY:=300;
        pCurrent.trans:=[-1*CurrentX,CurrentY,WorkZ];
        pCurrent.rot:=OrientZYX(0,0,180);
        pCurrent.robconf:=[1,0,-2,0];
        CalcTrack:=Bed1Wyong.uframe.trans.x+pCurrent.trans.x;
        IF CurrentY<1000 THEN CalcTrack:=CalcTrack+1200; ENDIF
        IF CalcTrack<TrackMin THEN CalcTrack:=TrackMin; ENDIF
        IF CalcTrack>TrackMax THEN CalcTrack:=TrackMax; ENDIF
        pCurrent.extax:=[CalcTrack,9E+09,9E+09,9E+09,9E+09,9E+09];
        MoveL pCurrent,vTravel,fine,tHeli\WObj:=Bed1Wyong;

        ! Point 17: (1130, 300) [work]
        CurrentX:=1130;
        CurrentY:=300;
        pCurrent.trans:=[-1*CurrentX,CurrentY,WorkZ];
        pCurrent.rot:=OrientZYX(0,0,180);
        pCurrent.robconf:=[1,0,-2,0];
        CalcTrack:=Bed1Wyong.uframe.trans.x+pCurrent.trans.x;
        IF CurrentY<1000 THEN CalcTrack:=CalcTrack+1200; ENDIF
        IF CalcTrack<TrackMin THEN CalcTrack:=TrackMin; ENDIF
        IF CalcTrack>TrackMax THEN CalcTrack:=TrackMax; ENDIF
        pCurrent.extax:=[CalcTrack,9E+09,9E+09,9E+09,9E+09,9E+09];
        MoveL pCurrent,vTravel,fine,tHeli\WObj:=Bed1Wyong;

        ! Point 18: (1130, 1550) [work]
        CurrentX:=1130;
        CurrentY:=1550;
        pCurrent.trans:=[-1*CurrentX,CurrentY,WorkZ];
        pCurrent.rot:=OrientZYX(0,0,180);
        pCurrent.robconf:=[1,0,-2,0];
        CalcTrack:=Bed1Wyong.uframe.trans.x+pCurrent.trans.x;
        IF CurrentY<1000 THEN CalcTrack:=CalcTrack+1200; ENDIF
        IF CalcTrack<TrackMin THEN CalcTrack:=TrackMin; ENDIF
        IF CalcTrack>TrackMax THEN CalcTrack:=TrackMax; ENDIF
        pCurrent.extax:=[CalcTrack,9E+09,9E+09,9E+09,9E+09,9E+09];
        MoveL pCurrent,vTravel,fine,tHeli\WObj:=Bed1Wyong;

        ! Point 19: (1430, 1550) [work]
        CurrentX:=1430;
        CurrentY:=1550;
        pCurrent.trans:=[-1*CurrentX,CurrentY,WorkZ];
        pCurrent.rot:=OrientZYX(0,0,180);
        pCurrent.robconf:=[1,0,-2,0];
        CalcTrack:=Bed1Wyong.uframe.trans.x+pCurrent.trans.x;
        IF CurrentY<1000 THEN CalcTrack:=CalcTrack+1200; ENDIF
        IF CalcTrack<TrackMin THEN CalcTrack:=TrackMin; ENDIF
        IF CalcTrack>TrackMax THEN CalcTrack:=TrackMax; ENDIF
        pCurrent.extax:=[CalcTrack,9E+09,9E+09,9E+09,9E+09,9E+09];
        MoveL pCurrent,vTravel,fine,tHeli\WObj:=Bed1Wyong;

